# B&R Automation Studio project OpcUaSample410_BrbLibUa103 (part 8)

#### BrbIsWithinRangeUdint.c - Gibt zurück, ob sich ein Wert innerhalb eines Bereichs befindet
```c
#include <bur/plctypes.h>
#ifdef __cplusplus
	extern "C"
	{
#endif

	#include "BrbLib.h"
	#include <AnsiCFunc.h>

#ifdef __cplusplus
	};
#endif

// NOLINTBEGIN(readability-*, bugprone-easily-swappable-parameters, clang-diagnostic-invalid-utf8, clang-diagnostic-invalid-source-encoding, clang-diagnostic-pointer-arith, clang-diagnostic-strict-prototypes, hicpp-uppercase-literal-suffix, cppcoreguidelines-*, performance-*)

/* Gibt zurück, ob sich ein Wert innerhalb eines Bereichs befindet */
plcbit BrbIsWithinRangeUdint(unsigned long nValue, unsigned long nRangeMin, unsigned long nRangeMax, unsigned long nTolerance)
{
	BOOL bResult = 0;
	if(nRangeMin > nRangeMax)
	{
		UDINT nTemp = nRangeMin;
		nRangeMin = nRangeMax;
		nRangeMax = nTemp;
	}
	UDINT nMin = 0;
	if(nTolerance < nRangeMin)
	{
		nMin = nRangeMin - nTolerance;
	}
	UDINT nMax = nRangeMax + nTolerance;
	if(nValue >= nMin && nValue <= nMax)
	{
		bResult = 1;
	}
	return bResult;
}

// NOLINTEND(readability-*, bugprone-easily-swappable-parameters, clang-diagnostic-invalid-utf8, clang-diagnostic-invalid-source-encoding, clang-diagnostic-pointer-arith, clang-diagnostic-strict-prototypes, hicpp-uppercase-literal-suffix, cppcoreguidelines-*, performance-*)
```

#### BrbIsWithinRangeReal.c - Gibt zurück, ob sich ein Wert innerhalb eines Bereichs befindet
```c
#include <bur/plctypes.h>
#ifdef __cplusplus
	extern "C"
	{
#endif

	#include "BrbLib.h"
	#include <AnsiCFunc.h>

#ifdef __cplusplus
	};
#endif

// NOLINTBEGIN(readability-*, bugprone-easily-swappable-parameters, clang-diagnostic-invalid-utf8, clang-diagnostic-invalid-source-encoding, clang-diagnostic-pointer-arith, clang-diagnostic-strict-prototypes, hicpp-uppercase-literal-suffix, cppcoreguidelines-*, performance-*)

/* Gibt zurück, ob sich ein Wert innerhalb eines Bereichs befindet */
plcbit BrbIsWithinRangeReal(float rValue, float rRangeMin, float rRangeMax, float rTolerance)
{
	BOOL bResult = 0;
	if(rRangeMin > rRangeMax)
	{
		REAL nTemp = rRangeMin;
		rRangeMin = rRangeMax;
		rRangeMax = nTemp;
	}
	if(rTolerance < 0.0f)
	{
		rTolerance = rTolerance * -1.00000000000f;
	}
	REAL rMin = rRangeMin - rTolerance;
	REAL rMax = rRangeMax + rTolerance;
	if(rValue >= rMin && rValue <= rMax)
	{
		bResult = 1;
	}
	return bResult;
}

// NOLINTEND(readability-*, bugprone-easily-swappable-parameters, clang-diagnostic-invalid-utf8, clang-diagnostic-invalid-source-encoding, clang-diagnostic-pointer-arith, clang-diagnostic-strict-prototypes, hicpp-uppercase-literal-suffix, cppcoreguidelines-*, performance-*)
```

#### BrbIsWithinRangeLReal.c - Gibt zurück, ob sich ein Wert innerhalb eines Bereichs befindet
```c
#include <bur/plctypes.h>
#ifdef __cplusplus
	extern "C"
	{
#endif

	#include "BrbLib.h"
	#include <AnsiCFunc.h>

#ifdef __cplusplus
	};
#endif

// NOLINTBEGIN(readability-*, bugprone-easily-swappable-parameters, clang-diagnostic-invalid-utf8, clang-diagnostic-invalid-source-encoding, clang-diagnostic-pointer-arith, clang-diagnostic-strict-prototypes, hicpp-uppercase-literal-suffix, cppcoreguidelines-*, performance-*)

/* Gibt zurück, ob sich ein Wert innerhalb eines Bereichs befindet */
plcbit BrbIsWithinRangeLReal(double rValue, double rRangeMin, double rRangeMax, double rTolerance)
{
	BOOL bResult = 0;
	if(rRangeMin > rRangeMax)
	{
		LREAL nTemp = rRangeMin;
		rRangeMin = rRangeMax;
		rRangeMax = nTemp;
	}
	if(rTolerance < 0.0)
	{
		rTolerance = rTolerance*(LREAL)-1.00000000000;
	}
	LREAL rMin = rRangeMin - rTolerance;
	LREAL rMax = rRangeMax + rTolerance;
	if(rValue >= rMin && rValue <= rMax)
	{
		bResult = 1;
	}
	return bResult;
}

// NOLINTEND(readability-*, bugprone-easily-swappable-parameters, clang-diagnostic-invalid-utf8, clang-diagnostic-invalid-source-encoding, clang-diagnostic-pointer-arith, clang-diagnostic-strict-prototypes, hicpp-uppercase-literal-suffix, cppcoreguidelines-*, performance-*)
```

#### BrbGetAngleRad.c - Rechnet einen Winkel von Grad ins Bogenmass um
```c
/********************************************************************
 * COPYRIGHT -- Bernecker + Rainer
 ********************************************************************
 * Library: BrbLib
 * File: BrbGetAngleRad.c
 * Author: niedermeierr
 * Created: July 19, 2014
 ********************************************************************
 * Implementation of library BrbLib
 ********************************************************************/

#include <bur/plctypes.h>
#ifdef __cplusplus
	extern "C"
	{
#endif

#include "BrbLib.h"
#include <math.h>

#ifdef __cplusplus
	};
#endif

// NOLINTBEGIN(readability-*, bugprone-easily-swappable-parameters, clang-diagnostic-invalid-utf8, clang-diagnostic-invalid-source-encoding, clang-diagnostic-pointer-arith, clang-diagnostic-strict-prototypes, hicpp-uppercase-literal-suffix, cppcoreguidelines-*, performance-*)

/* Rechnet einen Winkel von Grad ins Bogenmass um */
float BrbGetAngleRad(float rAngleDeg)
{
	REAL nResult = rAngleDeg * rBRB_FACTOR_DEG_TO_RAD;
	return nResult;
}

// NOLINTEND(readability-*, bugprone-easily-swappable-parameters, clang-diagnostic-invalid-utf8, clang-diagnostic-invalid-source-encoding, clang-diagnostic-pointer-arith, clang-diagnostic-strict-prototypes, hicpp-uppercase-literal-suffix, cppcoreguidelines-*, performance-*)
```

#### BrbGetAngleDeg.c - Rechnet einen Winkel vom Bogenmass in Grad um
```c
/********************************************************************
 * COPYRIGHT -- Bernecker + Rainer
 ********************************************************************
 * Library: BrbLib
 * File: BrbGetAngleDeg.c
 * Author: niedermeierr
 * Created: July 19, 2014
 ********************************************************************
 * Implementation of library BrbLib
 ********************************************************************/

#include <bur/plctypes.h>
#ifdef __cplusplus
	extern "C"
	{
#endif

#include "BrbLib.h"
#include <math.h>

#ifdef __cplusplus
	};
#endif

// NOLINTBEGIN(readability-*, bugprone-easily-swappable-parameters, clang-diagnostic-invalid-utf8, clang-diagnostic-invalid-source-encoding, clang-diagnostic-pointer-arith, clang-diagnostic-strict-prototypes, hicpp-uppercase-literal-suffix, cppcoreguidelines-*, performance-*)

/* Rechnet einen Winkel vom Bogenmass in Grad um */
float BrbGetAngleDeg(float rAngleRad)
{
	REAL nResult = rAngleRad * rBRB_FACTOR_RAD_TO_DEG;
	return nResult;
}

// NOLINTEND(readability-*, bugprone-easily-swappable-parameters, clang-diagnostic-invalid-utf8, clang-diagnostic-invalid-source-encoding, clang-diagnostic-pointer-arith, clang-diagnostic-strict-prototypes, hicpp-uppercase-literal-suffix, cppcoreguidelines-*, performance-*)
```

#### BrbNormalizeAngleRad.c - Normalisiert einen Bogenmasswinkel in den Bereich 0..2Pi
```c
/********************************************************************
 * COPYRIGHT -- Bernecker + Rainer
 ********************************************************************
 * Library: BrbLib
 * File: BrbNormalizeAngleRad.c
 * Author: niedermeierr
 * Created: September 05, 2014
 ********************************************************************
 * Implementation of library BrbLib
 ********************************************************************/

#include <bur/plctypes.h>
#ifdef __cplusplus
	extern "C"
	{
#endif

#include "BrbLib.h"
#include <AnsiCFunc.h>

#ifdef __cplusplus
	};
#endif

// NOLINTBEGIN(readability-*, bugprone-easily-swappable-parameters, clang-diagnostic-invalid-utf8, clang-diagnostic-invalid-source-encoding, clang-diagnostic-pointer-arith, clang-diagnostic-strict-prototypes, hicpp-uppercase-literal-suffix, cppcoreguidelines-*, performance-*)

/* Normalisiert einen Bogenmass-Winkel in den Bereich 0..2Pi */
float BrbNormalizeAngleRad(float rAngleRad)
{
	REAL rResult = 0.0f;
	DINT nMod = (DINT)(rAngleRad / 6.283185307179586476925286766559f);
	rResult = rAngleRad - ((REAL)nMod * 6.283185307179586476925286766559f);
	if(BrbIsNearlyZeroReal(rResult, 0.00017453292519943f))
	{
		// ~= 0.0
		rResult = 0.0f;
	}
	else if(rResult < 0.0f)
	{
		rResult += 6.283185307179586476925286766559f;
	}
	return rResult;
}

// NOLINTEND(readability-*, bugprone-easily-swappable-parameters, clang-diagnostic-invalid-utf8, clang-diagnostic-invalid-source-encoding, clang-diagnostic-pointer-arith, clang-diagnostic-strict-prototypes, hicpp-uppercase-literal-suffix, cppcoreguidelines-*, performance-*)
```

#### BrbNormalizeAngleDeg.c - Normalisiert einen Grad-Winkel in den Bereich 0..360°
```c
/********************************************************************
 * COPYRIGHT -- Bernecker + Rainer
 ********************************************************************
 * Library: BrbLib
 * File: BrbNormalizeAngleDeg.c
 * Author: niedermeierr
 * Created: September 05, 2014
 ********************************************************************
 * Implementation of library BrbLib
 ********************************************************************/

#include <bur/plctypes.h>
#ifdef __cplusplus
	extern "C"
	{
#endif

	#include "BrbLib.h"

#ifdef __cplusplus
	};
#endif

// NOLINTBEGIN(readability-*, bugprone-easily-swappable-parameters, clang-diagnostic-invalid-utf8, clang-diagnostic-invalid-source-encoding, clang-diagnostic-pointer-arith, clang-diagnostic-strict-prototypes, hicpp-uppercase-literal-suffix, cppcoreguidelines-*, performance-*)

/* Normalisiert einen Grad-Winkel in den Bereich 0..360° */
float BrbNormalizeAngleDeg(float rAngleDeg, plcbit bKeep360)
{
	REAL rResult = rBRB_DEGREE_0;
	if(bKeep360 == 1 && rAngleDeg == rBRB_DEGREE_360)
	{
		// 360.0° ist eigentlich 0°. Diese Korrektur kann hier verhindert werden.
		rResult = rBRB_DEGREE_360;
	}
	else
	{
		DINT nMod = (DINT)(rAngleDeg / rBRB_DEGREE_360);
		rResult = rAngleDeg - ((REAL)nMod * rBRB_DEGREE_360);
		if(rResult < rBRB_DEGREE_0)
		{
			rResult += rBRB_DEGREE_360;
		}
	}
	return rResult;
}

// NOLINTEND(readability-*, bugprone-easily-swappable-parameters, clang-diagnostic-invalid-utf8, clang-diagnostic-invalid-source-encoding, clang-diagnostic-pointer-arith, clang-diagnostic-strict-prototypes, hicpp-uppercase-literal-suffix, cppcoreguidelines-*, performance-*)
```

#### BrbIsWithinRangeAngle.c - Gibt zurück, ob sich ein Winkel innerhalb eines Bereichs befindet
```c
#include <bur/plctypes.h>
#ifdef __cplusplus
	extern "C"
	{
#endif

#include "BrbLib.h"

#ifdef __cplusplus
	};
#endif

// NOLINTBEGIN(readability-*, bugprone-easily-swappable-parameters, clang-diagnostic-invalid-utf8, clang-diagnostic-invalid-source-encoding, clang-diagnostic-pointer-arith, clang-diagnostic-strict-prototypes, hicpp-uppercase-literal-suffix, cppcoreguidelines-*, performance-*)

/* Gibt zurück, ob sich ein Winkel innerhalb eines Bereichs befindet */
plcbit BrbIsWithinRangeAngle(double rAngleAct, double rAngleStart, double rAngleEnd)
{
	BOOL bResult = 0;
	if(rAngleStart <= rAngleEnd)
	{
		if(rAngleAct >= rAngleStart && rAngleAct <= rAngleEnd)
		{
			bResult = 1;
		}
	}
	else
	{
		if(rAngleAct >= rAngleStart || rAngleAct <= rAngleEnd)
		{
			bResult = 1;
		}
	}
	return bResult;
}

// NOLINTEND(readability-*, bugprone-easily-swappable-parameters, clang-diagnostic-invalid-utf8, clang-diagnostic-invalid-source-encoding, clang-diagnostic-pointer-arith, clang-diagnostic-strict-prototypes, hicpp-uppercase-literal-suffix, cppcoreguidelines-*, performance-*)
```

#### BrbDetectAngleTransition.c - Erkennt eine Winkel-Übergang
```c
#include <bur/plctypes.h>
#ifdef __cplusplus
	extern "C"
	{
#endif

#include "BrbLib.h"

#ifdef __cplusplus
	};
#endif

// NOLINTBEGIN(readability-*, bugprone-easily-swappable-parameters, clang-diagnostic-invalid-utf8, clang-diagnostic-invalid-source-encoding, clang-diagnostic-pointer-arith, clang-diagnostic-strict-prototypes, hicpp-uppercase-literal-suffix, cppcoreguidelines-*, performance-*)

/* Erkennt den Übergang einer bestimmten Position bei einer 360°-Rundachse */
plcbit BrbDetectAngleTransition(double rTransPosition, plcbit bDirection, double rPosAct, double rPosOld)
{
	BOOL bResult = 0;
	// Richtung feststellen
	LREAL rDir =  rPosAct - rPosOld;
	if(rPosAct >= rBRB_DEGREE_0 && rPosAct <= rBRB_DEGREE_90 && rPosOld >= rBRB_DEGREE_270 && rPosOld <= rBRB_DEGREE_360)
	{
		// Übergang von 360° auf 0°
		rDir = +1.0;
	}
	else if(rPosAct >= rBRB_DEGREE_270 && rPosAct <= rBRB_DEGREE_360 && rPosOld >= rBRB_DEGREE_0 && rPosOld <= rBRB_DEGREE_90)
	{
		// Übergang von 0° auf 360°
		rDir = -1.0;
	}
	if(rTransPosition <= rBRB_DEGREE_90)
	{
		// Positionen um 90° nach positiv verschieben, um Übergang von 360° auf 0° zu vermeiden
		rTransPosition = (LREAL)BrbNormalizeAngleDeg((REAL)rTransPosition + rBRB_DEGREE_90, 0);
		rPosAct = (LREAL)BrbNormalizeAngleDeg((REAL)rPosAct + rBRB_DEGREE_90, 0);
		rPosOld = (LREAL)BrbNormalizeAngleDeg((REAL)rPosOld + rBRB_DEGREE_90, 0);
	}
	else if(rTransPosition >= rBRB_DEGREE_270)
	{
		// Positionen um 90° nach negativ verschieben, um Übergang von 360° auf 0° zu vermeiden
		rTransPosition = (LREAL)BrbNormalizeAngleDeg((REAL)rTransPosition - rBRB_DEGREE_90, 0);
		rPosAct = (LREAL)BrbNormalizeAngleDeg((REAL)rPosAct - rBRB_DEGREE_90, 0);
		rPosOld = (LREAL)BrbNormalizeAngleDeg((REAL)rPosOld - rBRB_DEGREE_90, 0);
	}
	// NOLINTBEGIN(bugprone-branch-clone)
	if(bDirection == 0 && rDir < rBRB_DEGREE_0)
	{
		// Negative Richtung
		if(rPosOld > rTransPosition && rPosAct <= rTransPosition)
		{
			bResult = 1;
		}
		else if(rPosOld >= rTransPosition && rPosAct < rTransPosition)
		{
			bResult = 1;
		}
	}
	else if(bDirection == 1 && rDir > rBRB_DEGREE_0)
	{
		// Positive Richtung
		if(rPosOld < rTransPosition && rPosAct >= rTransPosition)
		{
			bResult = 1;
		}
		else if(rPosOld <= rTransPosition && rPosAct > rTransPosition)
		{
			bResult = 1;
		}
	}
	// NOLINTEND(bugprone-branch-clone)
	return bResult;
}

// NOLINTEND(readability-*, bugprone-easily-swappable-parameters, clang-diagnostic-invalid-utf8, clang-diagnostic-invalid-source-encoding, clang-diagnostic-pointer-arith, clang-diagnostic-strict-prototypes, hicpp-uppercase-literal-suffix, cppcoreguidelines-*, performance-*)
```

#### BrbGetDistance2d.c - Errechnet die Distanz zwischen zwei Punkten
```c
#include <bur/plctypes.h>
#ifdef __cplusplus
	extern "C"
	{
#endif

	#include "BrbLib.h"
	#include <math.h>

#ifdef __cplusplus
	};
#endif

// NOLINTBEGIN(readability-*, bugprone-easily-swappable-parameters, clang-diagnostic-invalid-utf8, clang-diagnostic-invalid-source-encoding, clang-diagnostic-pointer-arith, clang-diagnostic-strict-prototypes, hicpp-uppercase-literal-suffix, cppcoreguidelines-*, performance-*)

/* Gibt die Distanz zwischen zwei Punkten im 2-dimensionalen Raum zurück */
double BrbGetDistance2d(double rX1, double rY1, double rX2, double rY2)
{
	return sqrt(pow((rX1-rX2), 2) + pow((rY1-rY2), 2));
}

// NOLINTEND(readability-*, bugprone-easily-swappable-parameters, clang-diagnostic-invalid-utf8, clang-diagnostic-invalid-source-encoding, clang-diagnostic-pointer-arith, clang-diagnostic-strict-prototypes, hicpp-uppercase-literal-suffix, cppcoreguidelines-*, performance-*)
```

#### BrbRoundDint.c - Rundet einen Dint
```c
/********************************************************************
 * COPYRIGHT -- Bernecker + Rainer
 ********************************************************************
 * Library: BrbLib
 * File: BrbRoundDint.c
 * Author: niedermeierr
 * Created: November 19, 2015
 ********************************************************************
 * Implementation of library BrbLib
 ********************************************************************/

#include <bur/plctypes.h>
#ifdef __cplusplus
	extern "C"
	{
#endif

#include "BrbLib.h"
#include <math.h>

#ifdef __cplusplus
	};
#endif

// NOLINTBEGIN(readability-*, bugprone-easily-swappable-parameters, clang-diagnostic-invalid-utf8, clang-diagnostic-invalid-source-encoding, clang-diagnostic-pointer-arith, clang-diagnostic-strict-prototypes, hicpp-uppercase-literal-suffix, cppcoreguidelines-*, performance-*)

/* Rundet einen Dint */
signed long BrbRoundDint(signed long nValue, enum BrbRound_ENUM eRound, unsigned char nDigits) // NOLINT(readability-function-cognitive-complexity)
{
	DINT nResult = nValue;
	if(nValue != 0)
	{
		if(nDigits < 1)
		{
			nDigits = 1;
		}
		BOOL bMinus = 0;
		if(nValue < 0)
		{
			bMinus = 1;
			nResult = nResult * -1;
			if(eRound == eBRB_ROUND_UP)
			{
				eRound = eBRB_ROUND_DOWN;
			}
			else if(eRound == eBRB_ROUND_DOWN)
			{
				eRound = eBRB_ROUND_UP;
			}
		}
		if(eRound == eBRB_ROUND_UP)
		{
			// Jede Stelle für sich runden
			USINT nDigit = 0;
			for(nDigit=1; nDigit<=nDigits; nDigit++)
			{
				DINT nDigitFactor = (DINT)pow(10, nDigit); // NOLINT(clang-diagnostic-bad-function-cast)
				DINT nNum0 = (DINT)((nResult / nDigitFactor) * nDigitFactor);
				DINT nRest = nResult - nNum0;
				if(nRest > 0)
				{
					nResult = nResult + (nDigitFactor - nRest);
				}
			}
		}
		else if(eRound == eBRB_ROUND_DOWN)
		{
			// Alle Rundungs-Stellen auf 0 setzen
			DINT nDigitFactor = (DINT)pow(10, nDigits); // NOLINT(clang-diagnostic-bad-function-cast)
			DINT nNum0 = (DINT)((nResult / nDigitFactor) * nDigitFactor);
			DINT nRest = nResult - nNum0;
			nResult = nResult - nRest;
		}
		else
		{
			DINT nDigitFactor = (DINT)pow(10.0, nDigits); // NOLINT(clang-diagnostic-bad-function-cast)
			DINT nNum0 = (DINT)(nResult / nDigitFactor);
			DINT nNum1 = nNum0 * nDigitFactor;
			DINT nRest = nResult - nNum1; // Rundungs-Stelle feststellen
			if(nRest >= 5 * (DINT)(nDigitFactor / 10.0))
			{
				nResult = BrbRoundDint(nResult, eBRB_ROUND_UP, nDigits);
			}
			else
			{
				nResult = BrbRoundDint(nResult, eBRB_ROUND_DOWN, nDigits);
			}
		}
		if(bMinus == 1)
		{
			nResult = nResult * -1;
		}
	}
	return nResult;
}

// NOLINTEND(readability-*, bugprone-easily-swappable-parameters, clang-diagnostic-invalid-utf8, clang-diagnostic-invalid-source-encoding, clang-diagnostic-pointer-arith, clang-diagnostic-strict-prototypes, hicpp-uppercase-literal-suffix, cppcoreguidelines-*, performance-*)
```

#### BrbScaleLReal.c - Skaliert ein analoges Eingangssignal linear auf einen Einheitswert
```c
/********************************************************************
 * COPYRIGHT -- Bernecker + Rainer
 ********************************************************************
 * Library: BrbLib
 * File: BrbScaleLReal.c
 * Author: niedermeierr
 * Created: October 11, 2021
 ********************************************************************
 * Implementation of library BrbLib
 ********************************************************************/

#include <bur/plctypes.h>
#ifdef __cplusplus
	extern "C"
	{
#endif

#include "BrbLib.h"

#ifdef __cplusplus
	};
#endif

// NOLINTBEGIN(readability-*, bugprone-easily-swappable-parameters, clang-diagnostic-invalid-utf8, clang-diagnostic-invalid-source-encoding, clang-diagnostic-pointer-arith, clang-diagnostic-strict-prototypes, hicpp-uppercase-literal-suffix, cppcoreguidelines-*, performance-*)

/* Skaliert ein analoges Signal linear */
double BrbScaleLReal(double rRaw, double rRawMin, double rRawMax, double rScaledMin, double rScaledMax, double rFactor, double rOffset)
{
	LREAL rResult = 0.0;
	LREAL rRawDiff = rRawMax - rRawMin;
	if(rRawDiff != 0.0) // Division durch 0 vermeiden
	{
		rResult = ((rScaledMin + ((rScaledMax - rScaledMin) / rRawDiff * (rRaw - rRawMin))) * rFactor) + rOffset;
	}
	return rResult;
}

// NOLINTEND(readability-*, bugprone-easily-swappable-parameters, clang-diagnostic-invalid-utf8, clang-diagnostic-invalid-source-encoding, clang-diagnostic-pointer-arith, clang-diagnostic-strict-prototypes, hicpp-uppercase-literal-suffix, cppcoreguidelines-*, performance-*)
```

#### BrbScaleAnalogInput.c - Skaliert ein analoges Eingangssignal linear auf einen Einheitswert
```c
/********************************************************************
 * COPYRIGHT -- Bernecker + Rainer
 ********************************************************************
 * Library: BrbLib
 * File: BrbScaleAnalogInput.c
 * Author: niedermeierr
 * Created: April 22, 2016
 ********************************************************************
 * Implementation of library BrbLib
 ********************************************************************/

#include <bur/plctypes.h>
#ifdef __cplusplus
	extern "C"
	{
#endif

#include "BrbLib.h"

#ifdef __cplusplus
	};
#endif

// NOLINTBEGIN(readability-*, bugprone-easily-swappable-parameters, clang-diagnostic-invalid-utf8, clang-diagnostic-invalid-source-encoding, clang-diagnostic-pointer-arith, clang-diagnostic-strict-prototypes, hicpp-uppercase-literal-suffix, cppcoreguidelines-*, performance-*)

/* Skaliert ein analoges Eingangssignal linear auf einen Einheitswert */
float BrbScaleAnalogInput(signed short nRaw, signed short nRawMin, signed short nRawMax, float rScaledMin, float rScaledMax, float rFactor, float rOffset)
{
	REAL rResult = 0.0f;
	DINT nRawDiff = nRawMax - nRawMin;
	if(nRawDiff != 0) // Division durch 0 vermeiden
	{
		rResult = ((rScaledMin + ((rScaledMax - rScaledMin) / (REAL)nRawDiff * (REAL)(nRaw - nRawMin))) * rFactor) + rOffset;
	}
	return rResult;
}

// NOLINTEND(readability-*, bugprone-easily-swappable-parameters, clang-diagnostic-invalid-utf8, clang-diagnostic-invalid-source-encoding, clang-diagnostic-pointer-arith, clang-diagnostic-strict-prototypes, hicpp-uppercase-literal-suffix, cppcoreguidelines-*, performance-*)
```

#### BrbScaleAnalogOutput.c - Skaliert ein analoges Ausgangssignal von einem EInheitswert
```c
/********************************************************************
 * COPYRIGHT -- Bernecker + Rainer
 ********************************************************************
 * Library: BrbLib
 * File: BrbScaleAnalogOutput.c
 * Author: niedermeierr
 * Created: April 22, 2016
 ********************************************************************
 * Implementation of library BrbLib
 ********************************************************************/

#include <bur/plctypes.h>
#ifdef __cplusplus
	extern "C"
	{
#endif

#include "BrbLib.h"

#ifdef __cplusplus
	};
#endif

// NOLINTBEGIN(readability-*, bugprone-easily-swappable-parameters, clang-diagnostic-invalid-utf8, clang-diagnostic-invalid-source-encoding, clang-diagnostic-pointer-arith, clang-diagnostic-strict-prototypes, hicpp-uppercase-literal-suffix, cppcoreguidelines-*, performance-*)

/* Skaliert ein analoges Ausgangssignal von einem Einheitswert */
signed short BrbScaleAnalogOutput(float rScaled, signed short nRawMin, signed short nRawMax, float rScaledMin, float rScaledMax, float rFactor, float rOffset)
{
	INT nResult = 0;
	REAL rScaleDiff = (rScaledMax - rScaledMin);
	if(rFactor != 0.0f && rScaleDiff != 0.0f) // Division durch 0 vermeiden // NOLINT(clang-diagnostic-float-equal)
	{
		REAL rRawMin = (REAL)nRawMin;
		REAL rRawMax = (REAL)nRawMax;
		REAL rValue = ((((rScaled - rOffset) / rFactor) - rScaledMin) * (rRawMax - rRawMin) / rScaleDiff) + rRawMin;
		if(rValue < rRawMin)
		{
			nResult = nRawMin;
		}
		else if(rValue > rRawMax)
		{
			nResult = nRawMax;
		}
		else
		{
			nResult = (INT)rValue;
		}
	}
	return nResult;
}

// NOLINTEND(readability-*, bugprone-easily-swappable-parameters, clang-diagnostic-invalid-utf8, clang-diagnostic-invalid-source-encoding, clang-diagnostic-pointer-arith, clang-diagnostic-strict-prototypes, hicpp-uppercase-literal-suffix, cppcoreguidelines-*, performance-*)
```

#### Package Logical/Libraries/BrbLib/Random - Erzeugung von Zufalls-Werten

#### BrbGetRandomPercent.c - Erzeugt eine Zufallszahl zwischen 0.0 und 1.0
```c
/********************************************************************
 * COPYRIGHT -- Bernecker + Rainer
 ********************************************************************
 * Library: BrbLib
 * File: BrbGetRandomPercent.c
 * Author: niedermeierr
 * Created: June 11, 2013
 ********************************************************************
 * Implementation of library BrbLib
 ********************************************************************/

#include <bur/plctypes.h>
#ifdef __cplusplus
	extern "C"
	{
#endif

#include "BrbLib.h"
#include "AnsiCFunc.h"

#ifdef __cplusplus
	};
#endif

// NOLINTBEGIN(readability-*, bugprone-easily-swappable-parameters, clang-diagnostic-invalid-utf8, clang-diagnostic-invalid-source-encoding, clang-diagnostic-pointer-arith, clang-diagnostic-strict-prototypes, hicpp-uppercase-literal-suffix, cppcoreguidelines-*, performance-*)

/* Erzeugt eine Zufallszahl zwischen 0.0 und 1.0 */
float BrbGetRandomPercent()
{
	INT	 	nRandom1 = (INT)rand(); // NOLINT(cert-msc30-c,cert-msc50-cpp, concurrency-mt-unsafe)
	DINT	nRandom2 = (DINT)nRandom1 + 32768;
	REAL	rRandom3 = (REAL)nRandom2 / 65535.0f;
	return rRandom3;
}

// NOLINTEND(readability-*, bugprone-easily-swappable-parameters, clang-diagnostic-invalid-utf8, clang-diagnostic-invalid-source-encoding, clang-diagnostic-pointer-arith, clang-diagnostic-strict-prototypes, hicpp-uppercase-literal-suffix, cppcoreguidelines-*, performance-*)
```

#### BrbGetRandomBool.c - Erzeugt einen boolschen Zufallswert
```c
/********************************************************************
 * COPYRIGHT -- Bernecker + Rainer
 ********************************************************************
 * Library: BrbLib
 * File: BrbGetRandomBool.c
 * Author: niedermeierr
 * Created: June 11, 2013
 ********************************************************************
 * Implementation of library BrbLib
 ********************************************************************/

#include <bur/plctypes.h>
#ifdef __cplusplus
	extern "C"
	{
#endif

#include "BrbLib.h"

#ifdef __cplusplus
	};
#endif

// NOLINTBEGIN(readability-*, bugprone-easily-swappable-parameters, clang-diagnostic-invalid-utf8, clang-diagnostic-invalid-source-encoding, clang-diagnostic-pointer-arith, clang-diagnostic-strict-prototypes, hicpp-uppercase-literal-suffix, cppcoreguidelines-*, performance-*)

/* Erzeugt einen boolschen Zufallswert */
plcbit BrbGetRandomBool()
{
	BOOL bRandom = (BOOL)(BrbGetRandomPercent()*(2));
	return bRandom;
}

// NOLINTEND(readability-*, bugprone-easily-swappable-parameters, clang-diagnostic-invalid-utf8, clang-diagnostic-invalid-source-encoding, clang-diagnostic-pointer-arith, clang-diagnostic-strict-prototypes, hicpp-uppercase-literal-suffix, cppcoreguidelines-*, performance-*)
```

#### BrbGetRandomUdint.c - Erzeugt eine Zufallszahl zwischen nMin und nMax
```c
/********************************************************************
 * COPYRIGHT -- Bernecker + Rainer
 ********************************************************************
 * Library: BrbLib
 * File: BrbGetRandomUdint.c
 * Author: niedermeierr
 * Created: June 11, 2013
 ********************************************************************
 * Implementation of library BrbLib
 ********************************************************************/

#include <bur/plctypes.h>
#ifdef __cplusplus
	extern "C"
	{
#endif

#include "BrbLib.h"

#ifdef __cplusplus
	};
#endif

// NOLINTBEGIN(readability-*, bugprone-easily-swappable-parameters, clang-diagnostic-invalid-utf8, clang-diagnostic-invalid-source-encoding, clang-diagnostic-pointer-arith, clang-diagnostic-strict-prototypes, hicpp-uppercase-literal-suffix, cppcoreguidelines-*, performance-*)

/* Erzeugt eine Zufallszahl zwischen nMin und nMax */
unsigned long BrbGetRandomUdint(unsigned long nMin, unsigned long nMax)
{
	UDINT nRandom = 0;
	if(nMin == 0 && nMax == nBRB_UDINT_MAX)
	{
		nRandom = (UDINT)(BrbGetRandomPercent() * (REAL)nMax);
	}
	else
	{
		// Eigentlich ohne +1, aber dann ist es sehr unwahrscheinlich, dass sich der Max-Wert ergibt (RandomPercent muss 1.0 sein).
		// Das +1 erhöht die Chance dazu, muss dann aber korrigiert werden.
		nRandom = (UDINT)(BrbGetRandomPercent()*(REAL)(nMax-nMin+1))+nMin;
		if(nRandom > nMax)
		{
			nRandom = nMax;
		}
		else if(nMin > 0 && nMax == nBRB_UDINT_MAX && nRandom == 0)
		{
			nRandom = nBRB_UDINT_MAX;
		}
	}
	return nRandom;
}

// NOLINTEND(readability-*, bugprone-easily-swappable-parameters, clang-diagnostic-invalid-utf8, clang-diagnostic-invalid-source-encoding, clang-diagnostic-pointer-arith, clang-diagnostic-strict-prototypes, hicpp-uppercase-literal-suffix, cppcoreguidelines-*, performance-*)
```

#### BrbGetRandomDint.c - Erzeugt eine Zufallszahl zwischen nMin und nMax
```c
/********************************************************************
 * COPYRIGHT -- Bernecker + Rainer
 ********************************************************************
 * Library: BrbLib
 * File: BrbGetRandomDint.c
 * Author: niedermeierr
 * Created: June 11, 2013
 ********************************************************************
 * Implementation of library BrbLib
 ********************************************************************/

#include <bur/plctypes.h>
#ifdef __cplusplus
	extern "C"
	{
#endif

#include "BrbLib.h"
#include <AnsiCFunc.h>

#ifdef __cplusplus
	};
#endif

// NOLINTBEGIN(readability-*, bugprone-easily-swappable-parameters, clang-diagnostic-invalid-utf8, clang-diagnostic-invalid-source-encoding, clang-diagnostic-pointer-arith, clang-diagnostic-strict-prototypes, hicpp-uppercase-literal-suffix, cppcoreguidelines-*, performance-*)

/* Erzeugt eine Zufallszahl zwischen nMin und nMax */
signed long BrbGetRandomDint(signed long nMin, signed long nMax)
{
	DINT nRandom = 0;
	if(nMin >= 0 && nMax >= 0)
	{
		nRandom = (DINT)BrbGetRandomUdint((UDINT)nMin, (UDINT)nMax);
	}
	else if(nMin < 0 && nMax < 0)
	{
		nRandom = (DINT)BrbGetRandomUdint((UDINT)abs(nMax), (UDINT)abs(nMin));
		nRandom = nRandom * -1;
	}
	else
	{
		// Eigentlich ohne +2.0, aber dann ist es sehr unwahrscheinlich, dass sich der Max-Wert ergibt (RandomPercent muss 1.0 sein).
		// Das +2.0 erhöht die Chance dazu, muss dann aber korrigiert werden.
		LREAL rRange = (LREAL)nMax - (LREAL)nMin + (LREAL)2.0;
		REAL rRangeRandom = BrbGetRandomPercent() * (REAL)rRange;
		LREAL rRandom = (LREAL)rRangeRandom + (LREAL)nMin - (LREAL)1.0;
		nRandom = (DINT)rRandom;
		// NOLINTBEGIN(bugprone-branch-clone)
		if(nRandom > nMax)
		{
			nRandom = nMax;
		}
		else if(nMin > 0 && nMax == nBRB_DINT_MAX && nRandom == 0)
		{
			nRandom = nMax;
		}
		else if(nRandom < nMin)
		{
			nRandom = nMin;
		}
		// NOLINTEND(bugprone-branch-clone)
	}
	return nRandom;
}

// NOLINTEND(readability-*, bugprone-easily-swappable-parameters, clang-diagnostic-invalid-utf8, clang-diagnostic-invalid-source-encoding, clang-diagnostic-pointer-arith, clang-diagnostic-strict-prototypes, hicpp-uppercase-literal-suffix, cppcoreguidelines-*, performance-*)
```

#### BrbGetRandomText.c - Erzeugt einen Zufallstext mit bestimmter Länge (nur Zahlen, Groß- und Kleinbuchstaben)
```c
#include <bur/plctypes.h>
#ifdef __cplusplus
	extern "C"
	{
#endif
	#include "BrbLib.h"
#include <string.h>

#ifdef __cplusplus
	};
#endif

// NOLINTBEGIN(readability-*, bugprone-easily-swappable-parameters, clang-diagnostic-invalid-utf8, clang-diagnostic-invalid-source-encoding, clang-diagnostic-pointer-arith, clang-diagnostic-strict-prototypes, hicpp-uppercase-literal-suffix, cppcoreguidelines-*, performance-*)

/* Erzeugt einen Zufallstext mit bestimmter Länge (nur Zahlen, Groß- und Kleinbuchstaben) */
unsigned long BrbGetRandomText(plcstring* pText, unsigned long nTextSize, unsigned long nTextLength)
{
	memset(pText, 0, nTextSize);
	if(nTextLength >= nTextSize)
	{
		nTextLength = nTextSize-1;
	}
	UDINT nCharIndex = 0;
	for(nCharIndex=0; nCharIndex<nTextLength; nCharIndex++)
	{
		USINT nChar = 0;
		DINT nBlockIndex = BrbGetRandomDint(0,2);
		if (nBlockIndex == 0)
		{
			// Zahl
			nChar = (USINT)BrbGetRandomUdint(48,57);
		}
		else if (nBlockIndex == 1)
		{
			// Großbuchstabe
			nChar = (USINT)BrbGetRandomUdint(65,90);
		}
		else
		{
			// KLeinbuchstabe
			nChar = (USINT)BrbGetRandomUdint(97,122);
		}
		USINT* pChar = (USINT*)pText + nCharIndex;
		*pChar = nChar;
	}
	return nTextLength;
}

// NOLINTEND(readability-*, bugprone-easily-swappable-parameters, clang-diagnostic-invalid-utf8, clang-diagnostic-invalid-source-encoding, clang-diagnostic-pointer-arith, clang-diagnostic-strict-prototypes, hicpp-uppercase-literal-suffix, cppcoreguidelines-*, performance-*)
```

#### BrbGetRandomString.c - Erzeugt einen Zufallstext mit bestimmter Länge aus einer Blockauswahl
```c
#include <bur/plctypes.h>
#ifdef __cplusplus
	extern "C"
	{
#endif
	#include "BrbLib.h"
	#include <string.h>

#ifdef __cplusplus
	};
#endif

// NOLINTBEGIN(readability-*, bugprone-easily-swappable-parameters, clang-diagnostic-invalid-utf8, clang-diagnostic-invalid-source-encoding, clang-diagnostic-pointer-arith, clang-diagnostic-strict-prototypes, hicpp-uppercase-literal-suffix, cppcoreguidelines-*, performance-*)

/* Erzeugt einen Zufallstext mit bestimmter Länge aus einer Zeichenblockauswahl */
unsigned long BrbGetRandomString(plcstring* pText, unsigned long nTextSize, unsigned long nTextLength, enum BrbRandomString_ENUM eSelection)
{
	USINT anSelection[256];
	memset((USINT*)&anSelection, 0, sizeof(anSelection));
	UINT nChar = 0;
	UINT nSelectionLength = 0;
	if((eSelection & eBRB_RANDOM_STRING_NUMBERS) == eBRB_RANDOM_STRING_NUMBERS) // NOLINT(hicpp-signed-bitwise)
	{
		// 0123456789
		for(nChar=48;nChar<=57;nChar++)
		{
			anSelection[nSelectionLength] = (USINT)nChar;
			nSelectionLength++;
		}
	}
	if((eSelection & eBRB_RANDOM_STRING_UPPER_LETTERS) == eBRB_RANDOM_STRING_UPPER_LETTERS) // NOLINT(hicpp-signed-bitwise)
	{
		//ABCDEFGHIJKLMNOPQRSTUVWXYZ
		for(nChar=65;nChar<=90;nChar++)
		{
			anSelection[nSelectionLength] = (USINT)nChar;
			nSelectionLength++;
		}
	}
	if((eSelection & eBRB_RANDOM_STRING_LOWER_LETTERS) == eBRB_RANDOM_STRING_LOWER_LETTERS) // NOLINT(hicpp-signed-bitwise)
	{
		//abcdefghijklmnopqrstuvwxyz
		for(nChar=97;nChar<=122;nChar++)
		{
			anSelection[nSelectionLength] = (USINT)nChar;
			nSelectionLength++;
		}
	}
	if((eSelection & eBRB_RANDOM_STRING_SPACE) == eBRB_RANDOM_STRING_SPACE) // NOLINT(hicpp-signed-bitwise)
	{
		//" "
		anSelection[nSelectionLength] = 32;
		nSelectionLength++;
	}
	if((eSelection & eBRB_RANDOM_STRING_PUNCTUATION) == eBRB_RANDOM_STRING_PUNCTUATION) // NOLINT(hicpp-signed-bitwise)
	{
		//!"#$%&'()*+,-./
		for(nChar=33;nChar<=47;nChar++)
		{
			anSelection[nSelectionLength] = (USINT)nChar;
			nSelectionLength++;
		}
		//:;<=>?@
		for(nChar=58;nChar<=64;nChar++)
		{
			anSelection[nSelectionLength] = (USINT)nChar;
			nSelectionLength++;
		}
		//[\]^_`
		for(nChar=91;nChar<=96;nChar++)
		{
			anSelection[nSelectionLength] = (USINT)nChar;
			nSelectionLength++;
		}
		// {|}~
		for(nChar=123;nChar<=126;nChar++)
		{
			anSelection[nSelectionLength] = (USINT)nChar;
			nSelectionLength++;
		}
	}
	if((eSelection & eBRB_RANDOM_STRING_SYMBOLS) == eBRB_RANDOM_STRING_SYMBOLS) // NOLINT(hicpp-signed-bitwise)
	{
		for(nChar=128;nChar<=255;nChar++)
		{
			anSelection[nSelectionLength] = (USINT)nChar;
			nSelectionLength++;
		}
	}
	if((eSelection & eBRB_RANDOM_STRING_CONTROLCHARS) == eBRB_RANDOM_STRING_CONTROLCHARS) // NOLINT(hicpp-signed-bitwise)
	{
		// <127=DEL>
		anSelection[nSelectionLength] = 127;
		nSelectionLength++;
		// <1=SOH><2=STX><3=ETX><4=EOT><5=ENQ><6=ACK><7=BEL><8=BS><9=TAB><10=LF><11=VT><12=FF><13=CR><14=SO><15=SI><16=DLE>
		// <17=DC1><18=DC2><19=DC3><20=DC4><21=NAK><22=SYN><23=ETB><24=CAN><25=EM><26=SUB>27=ESC<28=FS><29=GS><30=RS><31=US>
		for(nChar=1;nChar<=31;nChar++)
		{
			anSelection[nSelectionLength] = (USINT)nChar;
			nSelectionLength++;
		}
	}
	return BrbGetRandomStringExt(pText, nTextSize, nTextLength, (STRING*)&anSelection);
}

// NOLINTEND(readability-*, bugprone-easily-swappable-parameters, clang-diagnostic-invalid-utf8, clang-diagnostic-invalid-source-encoding, clang-diagnostic-pointer-arith, clang-diagnostic-strict-prototypes, hicpp-uppercase-literal-suffix, cppcoreguidelines-*, performance-*)
```

#### BrbGetRandomStringExt.c - Erzeugt einen Zufallstext mit bestimmter Länge aus einer Zeichenauswahl
```c
#include <bur/plctypes.h>
#ifdef __cplusplus
	extern "C"
	{
#endif
	#include "BrbLib.h"
	#include <string.h>

#ifdef __cplusplus
	};
#endif

// NOLINTBEGIN(readability-*, bugprone-easily-swappable-parameters, clang-diagnostic-invalid-utf8, clang-diagnostic-invalid-source-encoding, clang-diagnostic-pointer-arith, clang-diagnostic-strict-prototypes, hicpp-uppercase-literal-suffix, cppcoreguidelines-*, performance-*)

/* Erzeugt einen Zufallstext mit bestimmter Länge aus einer Zeichenauswahl */
unsigned long BrbGetRandomStringExt(plcstring* pText, unsigned long nTextSize, unsigned long nTextLength, plcstring* pSelection)
{
	memset(pText, 0, nTextSize);
	UDINT nSelectionLength = strlen(pSelection);
	if(nSelectionLength > 0)
	{
		if(nTextLength >= nTextSize)
		{
			nTextLength = nTextSize-1;
		}
		UDINT nCharIndex = 0;
		for(nCharIndex=0; nCharIndex<nTextLength; nCharIndex++)
		{
			UDINT nSelectionCharIndex = BrbGetRandomUdint(0,nSelectionLength-1);
			USINT* pChar = (USINT*)pText + nCharIndex;
			*pChar = *((USINT*)pSelection + nSelectionCharIndex);
		}
	}
	else
	{
		nTextLength = 0;
	}
	return nTextLength;
}

// NOLINTEND(readability-*, bugprone-easily-swappable-parameters, clang-diagnostic-invalid-utf8, clang-diagnostic-invalid-source-encoding, clang-diagnostic-pointer-arith, clang-diagnostic-strict-prototypes, hicpp-uppercase-literal-suffix, cppcoreguidelines-*, performance-*)
```

#### Package Logical/Libraries/BrbLib/IpAndSubnet - Ip-Adress-Funktionen

#### BrbIpToNumericalArray.c - Wandelt eine Ip-Adresse in eine Byte-Array
```c
/********************************************************************
 * COPYRIGHT -- Bernecker + Rainer
 ********************************************************************
 * Library: BrbLib
 * File: BrbIpToNumericalArray.c
 * Author: niedermeierr
 * Created: July 05, 2022
 ********************************************************************
 * Implementation of library BrbLib
 ********************************************************************/

#include <bur/plctypes.h>
#ifdef __cplusplus
	extern "C"
	{
#endif

#include "BrbLib.h"
#include <string.h>

#ifdef __cplusplus
	};
#endif

// NOLINTBEGIN(readability-*, bugprone-easily-swappable-parameters, clang-diagnostic-invalid-utf8, clang-diagnostic-invalid-source-encoding, clang-diagnostic-pointer-arith, clang-diagnostic-strict-prototypes, hicpp-uppercase-literal-suffix, cppcoreguidelines-*, performance-*)

/* Wandelt eine textuelle Ip-Adresse in ein USINT-Array */
unsigned short BrbIpToNumericalArray(plcstring* pIp, unsigned long pUsintArray)
{
	// Prüfung der Parameter
	if(pIp == 0)
	{
		return eBRB_ERR_NULL_POINTER;
	}
	if(pUsintArray == 0)
	{
		return eBRB_ERR_NULL_POINTER;
	}
	// Die einzelnen Segemente in ein String-Array kopieren
	STRING asIp[4][nBRB_IP_ADR_CHAR_MAX];
	BrbStringSplitEmpty(pIp, ".", (UDINT)&asIp, 3, sizeof(asIp[0]));
	// Die einzelnen Segemente in USINT wandeln
	UINT nIndex = 0;
	for(nIndex=0; nIndex<=3; nIndex++)
	{
		*(((USINT*)pUsintArray)+nIndex) = (USINT)brsatoi((UDINT)&asIp[nIndex]);
	}
	return eBRB_ERR_OK;
}

// NOLINTEND(readability-*, bugprone-easily-swappable-parameters, clang-diagnostic-invalid-utf8, clang-diagnostic-invalid-source-encoding, clang-diagnostic-pointer-arith, clang-diagnostic-strict-prototypes, hicpp-uppercase-literal-suffix, cppcoreguidelines-*, performance-*)
```

#### BrbCheckIpAddress.c - Prüft eine Ip-Adresse und berichtigt sie gegebenenfalls
```c
/********************************************************************
 * COPYRIGHT -- Bernecker + Rainer
 ********************************************************************
 * Library: BrbLib
 * File: BrbCheckIpAddress.c
 * Author: niedermeierr
 * Created: November 25, 2014
 ********************************************************************
 * Implementation of library BrbLib
 ********************************************************************/

#include <bur/plctypes.h>
#ifdef __cplusplus
	extern "C"
	{
#endif

#include "BrbLib.h"
#include <string.h>

#ifdef __cplusplus
	};
#endif

// NOLINTBEGIN(readability-*, bugprone-easily-swappable-parameters, clang-diagnostic-invalid-utf8, clang-diagnostic-invalid-source-encoding, clang-diagnostic-pointer-arith, clang-diagnostic-strict-prototypes, hicpp-uppercase-literal-suffix, cppcoreguidelines-*, performance-*)

/* Prüft eine Ip-Adresse und berichtigt sie gegebenenfalls */
plcbit BrbCheckIpAddress(plcstring* pIpAddress)
{
	// Eine Ip-Adresse darf keine Buchstaben enthalten.
	// Die einzelnen Segmente dürfen keine führenden Nullen haben, weil sie sonst vom Betriebssystem als Oktal-Zahl erkannt werden.
	BOOL bResult = 0;
	STRING sAdr[4][nBRB_IP_ADR_CHAR_MAX];
	BrbStringSplitEmpty(pIpAddress, ".", (UDINT)&sAdr, 3, sizeof(sAdr[0]));
	UINT nIndex = 0;
	for(nIndex=0; nIndex<=3; nIndex++)
	{
		UDINT nLen = strlen(sAdr[nIndex]);
		if(nLen == 0)
		{
			// Leerstring wird zu "0"
			strcpy(sAdr[nIndex], "0");
		}
		else
		{
			// Nummern-Prüfung
			DINT nNumber = brsatoi((UDINT)&sAdr[nIndex]);
			nNumber = ((nNumber > 255)? 255 : ((nNumber < 0)? 0 : nNumber)); // auf 0..255 limitieren
			brsitoa(nNumber, (UDINT)&sAdr[nIndex]);
		}
	}
	// NOLINTBEGIN(clang-analyzer-security.insecureAPI.strcpy)
	strcpy(pIpAddress, "");
	strcat(pIpAddress, sAdr[0]);
	strcat(pIpAddress, ".");
	strcat(pIpAddress, sAdr[1]);
	strcat(pIpAddress, ".");
	strcat(pIpAddress, sAdr[2]);
	strcat(pIpAddress, ".");
	strcat(pIpAddress, sAdr[3]);
	// NOLINTEND(clang-analyzer-security.insecureAPI.strcpy)
	return bResult;
}

// NOLINTEND(readability-*, bugprone-easily-swappable-parameters, clang-diagnostic-invalid-utf8, clang-diagnostic-invalid-source-encoding, clang-diagnostic-pointer-arith, clang-diagnostic-strict-prototypes, hicpp-uppercase-literal-suffix, cppcoreguidelines-*, performance-*)
```

#### BrbCheckSubnet.c - Prüft eine Subnet-Maske
```c
/********************************************************************
 * COPYRIGHT -- Bernecker + Rainer
 ********************************************************************
 * Library: BrbLib
 * File: BrbCheckSubnet.c
 * Author: niedermeierr
 * Created: July 05, 2022
 ********************************************************************
 * Implementation of library BrbLib
 ********************************************************************/

#include <bur/plctypes.h>
#ifdef __cplusplus
	extern "C"
	{
#endif

#include "BrbLib.h"
#include <string.h>

#ifdef __cplusplus
	};
#endif

// NOLINTBEGIN(readability-*, bugprone-easily-swappable-parameters, clang-diagnostic-invalid-utf8, clang-diagnostic-invalid-source-encoding, clang-diagnostic-pointer-arith, clang-diagnostic-strict-prototypes, hicpp-uppercase-literal-suffix, cppcoreguidelines-*, performance-*)

/* Prüft eine Subnet-Angabe auf Gültigkeit */
plcbit BrbCheckSubnet(plcstring* pSubnet)
{
	BOOL bResult = 1;
	// Subnet in numerisches Array wandeln
	USINT anSubnet[4];	BrbIpToNumericalArray(pSubnet, (UDINT)&anSubnet);
	// Sobald eine Null im Bitmuster gesetzt ist, dürfen nur noch Nullen folgen
	UINT nIndex = 0;
	BOOL bFollowingBitsMustBeZero = 0;
	for(nIndex=0; nIndex<=3; nIndex++)
	{
		// Es dürfen nur bestimmte Bitmuster in einem Segment gesetzt sein (nur führende Einsen)
		// NOLINTBEGIN(bugprone-branch-clone)
		if(bFollowingBitsMustBeZero && anSubnet[nIndex] != 0)
		{
			// Keine führende 1
			bResult = 0;
			break;
		}
		else if(anSubnet[nIndex] == 255)
		{
			// Alle Bits des Netzwerk-Anteils gesetzt -> Passt
		}
		else if(anSubnet[nIndex] == 0
		|| anSubnet[nIndex] == 128	// #1000 0000
		|| anSubnet[nIndex] == 192	// #1100 0000
		|| anSubnet[nIndex] == 224	// #1110 0000
		|| anSubnet[nIndex] == 240	// #1111 0000
		|| anSubnet[nIndex] == 248	// #1111 1000
		|| anSubnet[nIndex] == 252	// #1111 1100
		|| anSubnet[nIndex] == 254	// #1111 1110
		)
		{
			// Nur führende Einsen -> Nachfolgende Segmente dürfen kein Bit gesetzt haben
			bFollowingBitsMustBeZero = 1;
		}
		else
		{
			// Keine führende 1
			bResult = 0;
			break;
		}
		// NOLINTEND(bugprone-branch-clone)
	}
	// Zusätzliche Prüfungen
	UDINT* pSubnetUdint = (UDINT*)&anSubnet; // NOLINT(clang-diagnostic-cast-align)
	if(*pSubnetUdint == 0)
	{
		// Nur Nullen sind nicht erlaubt
		bResult = 0;
	}
	if(*pSubnetUdint == nBRB_UDINT_MAX)
	{
		// Nur Einsen sind nicht erlaubt
		bResult = 0;
	}
	return bResult;
}

// NOLINTEND(readability-*, bugprone-easily-swappable-parameters, clang-diagnostic-invalid-utf8, clang-diagnostic-invalid-source-encoding, clang-diagnostic-pointer-arith, clang-diagnostic-strict-prototypes, hicpp-uppercase-literal-suffix, cppcoreguidelines-*, performance-*)
```

#### BrbGetIpAddressType.c - Gibt den Typ einer Ip-Adresse zurück
```c
/********************************************************************
 * COPYRIGHT -- Bernecker + Rainer
 ********************************************************************
 * Library: BrbLib
 * File: BrbGetIpAddressType.c
 * Author: niedermeierr
 * Created: July 05, 2022
 ********************************************************************
 * Implementation of library BrbLib
 ********************************************************************/

#include <bur/plctypes.h>
#ifdef __cplusplus
	extern "C"
	{
#endif

#include "BrbLib.h"
#include <string.h>

#ifdef __cplusplus
	};
#endif

// NOLINTBEGIN(readability-*, bugprone-easily-swappable-parameters, clang-diagnostic-invalid-utf8, clang-diagnostic-invalid-source-encoding, clang-diagnostic-pointer-arith, clang-diagnostic-strict-prototypes, hicpp-uppercase-literal-suffix, cppcoreguidelines-*, performance-*)

/* Gibt den Typen einer Ip-Adresse zurück (Netzwerk-oder Broadcast-Adresse) */
enum BrbIpAdrType_ENUM BrbGetIpAddressType(plcstring* pIp, plcstring* pSubnet)
{
	BrbIpAdrType_ENUM eResult = eBRB_IP_ADR_TYPE_UNKNOWN;
	// Ip und Subnet in numerische Arrays wandeln
	USINT anIp[4];			BrbIpToNumericalArray(pIp, (UDINT)&anIp);
	USINT anSubnet[4];	BrbIpToNumericalArray(pSubnet, (UDINT)&anSubnet);
	USINT anSubnetComplement[4];
	USINT anNetworkIp[4];
	USINT anBroadcastIp[4];
	UINT nIndex = 0;
	for(nIndex=0; nIndex<=3; nIndex++)
	{
		// Komplement des Subnets bilden (Bits umkehren), um so den Host-Anteil zu bekommen
		anSubnetComplement[nIndex] = ~anSubnet[nIndex];
		// Netzwerk-Adresse aufgrund des Subnets ermitteln (kleinste Adresse des Host-Bereichs)
		anNetworkIp[nIndex] = (anIp[nIndex] & anSubnet[nIndex]);
		// Broadcast-Adresse aufgrund des Subnets ermitteln (größte Adresse des Host-Bereichs)
		anBroadcastIp[nIndex] = (anIp[nIndex] & anSubnet[nIndex]) | anSubnetComplement[nIndex]; // NOLINT(hicpp-signed-bitwise)
	}
	// Vergleich mit den ermittelten Adressen
	UDINT* pIpUdint = (UDINT*)&anIp; // NOLINT(clang-diagnostic-cast-align)
	UDINT* pNetworkIpUdint = (UDINT*)&anNetworkIp; // NOLINT(clang-diagnostic-cast-align)
	UDINT* pBroadcastIpUdint = (UDINT*)&anBroadcastIp; // NOLINT(clang-diagnostic-cast-align)
	// Da auf direkte Gleichheit geprüft werden muss, können die 4 Byte-Segmente jeweils vereinfacht als UDINT (ebenfalls 4 Byte) verglichen werden
	// NOLINTBEGIN(bugprone-branch-clone)
	if(*pIpUdint == 0)
	{
		eResult = eBRB_IP_ADR_TYPE_UNKNOWN;
	}
	else if(*pIpUdint == nBRB_UDINT_MAX)
	{
		eResult = eBRB_IP_ADR_TYPE_UNKNOWN;
	}
	else if(*pIpUdint == *pNetworkIpUdint)
	{
		eResult = eBRB_IP_ADR_TYPE_NETWORK;
	}
	else if(*pIpUdint == *pBroadcastIpUdint)
	{
		eResult = eBRB_IP_ADR_TYPE_BROADCAST;
	}
	else
	{
		eResult = eBRB_IP_ADR_TYPE_HOST;
	}
	// NOLINTEND(bugprone-branch-clone)
	return eResult;
}

// NOLINTEND(readability-*, bugprone-easily-swappable-parameters, clang-diagnostic-invalid-utf8, clang-diagnostic-invalid-source-encoding, clang-diagnostic-pointer-arith, clang-diagnostic-strict-prototypes, hicpp-uppercase-literal-suffix, cppcoreguidelines-*, performance-*)
```

#### BrbCheckIpEqualSubnet.c - Prüft, ob sich zwei Ip-Adressen im selben Subnet befinden
```c
/********************************************************************
 * COPYRIGHT -- Bernecker + Rainer
 ********************************************************************
 * Library: BrbLib
 * File: BrbCheckIpEqualSubnet.c
 * Author: niedermeierr
 * Created: July 05, 2022
 ********************************************************************
 * Implementation of library BrbLib
 ********************************************************************/

#include <bur/plctypes.h>
#ifdef __cplusplus
	extern "C"
	{
#endif

#include "BrbLib.h"
#include <string.h>

#ifdef __cplusplus
	};
#endif

// NOLINTBEGIN(readability-*, bugprone-easily-swappable-parameters, clang-diagnostic-invalid-utf8, clang-diagnostic-invalid-source-encoding, clang-diagnostic-pointer-arith, clang-diagnostic-strict-prototypes, hicpp-uppercase-literal-suffix, cppcoreguidelines-*, performance-*)

/* Prüft, ob zwei Ip-Adressen im selben Subnet sind */
plcbit BrbCheckIpEqualSubnet(plcstring* pIp1, plcstring* pSubnet1, plcstring* pIp2, plcstring* pSubnet2)
{
	BOOL bResult = 1;
	// Ip's und Subnets in numerische Arrays wandeln
	USINT anIp1[4];			BrbIpToNumericalArray(pIp1, (UDINT)&anIp1);
	USINT anSubnet1[4];	BrbIpToNumericalArray(pSubnet1, (UDINT)&anSubnet1);
	USINT anIp2[4];			BrbIpToNumericalArray(pIp2, (UDINT)&anIp2);
	USINT anSubnet2[4];	BrbIpToNumericalArray(pSubnet2, (UDINT)&anSubnet2);
	// Vergleich der Netz-Anteile (durch Verundung mit dem Subnet wird der Host-Anteil elimniert)
	UINT nIndex = 0;
	for(nIndex=0; nIndex<=3; nIndex++)
	{
		// Subnet verodern (das Subnet gibt den Netz-Anteil an, somit wird der gemeinsame Netz-Anteil zum Vergleich verwendet)
		USINT nSubnet = anSubnet1[nIndex] | anSubnet2[nIndex];
		// Vergleich
		USINT nIp1 = anIp1[nIndex] & nSubnet;
		USINT nIp2 = anIp2[nIndex] & nSubnet;
		if(nIp1 != nIp2)
		{
			bResult = 0;
			break;
		}
	}
	return bResult;
}

// NOLINTEND(readability-*, bugprone-easily-swappable-parameters, clang-diagnostic-invalid-utf8, clang-diagnostic-invalid-source-encoding, clang-diagnostic-pointer-arith, clang-diagnostic-strict-prototypes, hicpp-uppercase-literal-suffix, cppcoreguidelines-*, performance-*)
```

#### Package Logical/Libraries/BrbLib/Additional - Erzeugung von Zufallszahlen

#### BrbDebounceInput.c - Entprellt einen Eingang
```c
/********************************************************************
 * COPYRIGHT -- Bernecker + Rainer
 ********************************************************************
 * Library: BrbLib
 * File: BrbDebounceInput.c
 * Author: niedermeierr
 * Created: April 15, 2015
 ********************************************************************
 * Implementation of library BrbLib
 ********************************************************************/

#include <bur/plctypes.h>
#ifdef __cplusplus
	extern "C"
	{
#endif

#include "BrbLib.h"

#ifdef __cplusplus
	};
#endif

// NOLINTBEGIN(readability-*, bugprone-easily-swappable-parameters, clang-diagnostic-invalid-utf8, clang-diagnostic-invalid-source-encoding, clang-diagnostic-pointer-arith, clang-diagnostic-strict-prototypes, hicpp-uppercase-literal-suffix, cppcoreguidelines-*, performance-*)

/* Entprellt einen Eingang */
void BrbDebounceInput(struct BrbDebounceInput* inst)
{
	inst->bOutput = 0;
	inst->fbDebounce.PT = (TIME)inst->nDebounceTime;
	TON(&inst->fbDebounce);
	if(inst->fbDebounce.Q == 1)
	{
		inst->fbDebounce.IN = 0;
		TON(&inst->fbDebounce);
	}
	if(inst->bInput == 1 && inst->fbDebounce.IN == 0)
	{
		inst->bOutput = 1;
		inst->fbDebounce.IN = 1;
		TON(&inst->fbDebounce);
	}
}

// NOLINTEND(readability-*, bugprone-easily-swappable-parameters, clang-diagnostic-invalid-utf8, clang-diagnostic-invalid-source-encoding, clang-diagnostic-pointer-arith, clang-diagnostic-strict-prototypes, hicpp-uppercase-literal-suffix, cppcoreguidelines-*, performance-*)
```

#### BrbGetStructMemberOffset.c - Gibt den Offset eines Struktur-Members zurück
```c
/********************************************************************
 * COPYRIGHT -- Bernecker + Rainer
 ********************************************************************
 * Library: BrbLib
 * File: BrbGetStructMemberOffset.c
 * Author: niedermeierr
 * Created: December 21, 2015
 ********************************************************************
 * Implementation of library BrbLib
 ********************************************************************/

#include <bur/plctypes.h>
#ifdef __cplusplus
	extern "C"
	{
#endif

#include "BrbLib.h"
#include <string.h>

#ifdef __cplusplus
	};
#endif

// NOLINTBEGIN(readability-*, bugprone-easily-swappable-parameters, clang-diagnostic-invalid-utf8, clang-diagnostic-invalid-source-encoding, clang-diagnostic-pointer-arith, clang-diagnostic-strict-prototypes, hicpp-uppercase-literal-suffix, cppcoreguidelines-*, performance-*)

/* Gibt den Offset eines Struktur-Members zurück */
unsigned short BrbGetStructMemberOffset(plcstring* pStructName, plcstring* pMemberName, unsigned long* pOffset)
{
	UINT nStatus = 0;
	*pOffset = 0;
	// Adresse der Struktur-Instanz ermitteln
	UDINT nAddressStruct = 0;
	UDINT nLen = 0;
	nStatus = PV_xgetadr((STRING*)pStructName, (UDINT*)&nAddressStruct, (UDINT*)&nLen);
	if(nStatus == 0)
	{
		// Adresse der Struktur-Member ermitteln
		UDINT nAddressMember = 0;
		STRING sMember[nBRB_PVNAME_CHAR_MAX];
		BrbStringCopy(sMember, pStructName, sizeof(sMember));
		BrbStringCat(sMember, ".", sizeof(sMember));
		BrbStringCat(sMember, pMemberName, sizeof(sMember));
		nStatus = PV_xgetadr((STRING*)&sMember, (UDINT*)&nAddressMember, (UDINT*)&nLen);
		if(nStatus == 0)
		{
			// Differenz ergibt Offset
			*pOffset = nAddressMember - nAddressStruct;
		}
	}
	return nStatus;
}

// NOLINTEND(readability-*, bugprone-easily-swappable-parameters, clang-diagnostic-invalid-utf8, clang-diagnostic-invalid-source-encoding, clang-diagnostic-pointer-arith, clang-diagnostic-strict-prototypes, hicpp-uppercase-literal-suffix, cppcoreguidelines-*, performance-*)
```

#### BrbGetCompilerVersion.c - Gibt die Version des Compilers zurück
```c
/********************************************************************
 * COPYRIGHT -- Bernecker + Rainer
 ********************************************************************
 * Library: BrbLib
 * File: BrbGetCompilerVersion.c
 * Author: niedermeierr
 * Created: October 24, 2019
 ********************************************************************
 * Implementation of library BrbLib
 ********************************************************************/

#include <bur/plctypes.h>
#ifdef __cplusplus
	extern "C"
	{
#endif

#include "BrbLib.h"
#include <string.h>

#ifdef __cplusplus
	};
#endif

// NOLINTBEGIN(readability-*, bugprone-easily-swappable-parameters, clang-diagnostic-invalid-utf8, clang-diagnostic-invalid-source-encoding, clang-diagnostic-pointer-arith, clang-diagnostic-strict-prototypes, hicpp-uppercase-literal-suffix, cppcoreguidelines-*, performance-*)

/* Gibt die Version des verwendeten GCC-Compilers zurück */
unsigned short BrbGetCompilerVersion(struct BrbCompilerVersion_TYP* pCompilerVersion)
{
	UINT nResult = 0;
	STRING sItoA[20];
	pCompilerVersion->bValid = 0;
	pCompilerVersion->nMajor = 0;
	pCompilerVersion->nMinor = 0;
	pCompilerVersion->nPatch = 0;
	pCompilerVersion->nTotal = 0;
	memset(&pCompilerVersion->sText, 0, sizeof(pCompilerVersion->sText));

	#ifdef __GNUC__
		pCompilerVersion->nMajor = __GNUC__;
		nResult += 4;
	#endif
	pCompilerVersion->nTotal += ((DINT)pCompilerVersion->nMajor * 10000);
	brsitoa((DINT)pCompilerVersion->nMajor, (UDINT)&sItoA);
	BrbStringCopy((STRING*)&pCompilerVersion->sText, sItoA, sizeof(pCompilerVersion->sText));
	BrbStringCat((STRING*)&pCompilerVersion->sText, ".", sizeof(pCompilerVersion->sText));

	#ifdef __GNUC_MINOR__
		pCompilerVersion->nMinor = __GNUC_MINOR__;
		nResult += 2;
	#endif
	pCompilerVersion->nTotal += ((DINT)pCompilerVersion->nMinor * 100);
	brsitoa((DINT)pCompilerVersion->nMinor, (UDINT)&sItoA);
	BrbStringCat((STRING*)&pCompilerVersion->sText, sItoA, sizeof(pCompilerVersion->sText));
	BrbStringCat((STRING*)&pCompilerVersion->sText, ".", sizeof(pCompilerVersion->sText));

	#ifdef __GNUC_PATCHLEVEL__
		pCompilerVersion->nPatch = __GNUC_PATCHLEVEL__;
		nResult += 1;
	#endif
	pCompilerVersion->nTotal += (DINT)pCompilerVersion->nPatch;
	brsitoa((DINT)pCompilerVersion->nPatch, (UDINT)&sItoA);
	BrbStringCat((STRING*)&pCompilerVersion->sText, sItoA, sizeof(pCompilerVersion->sText));

	if(nResult >= 7)
	{
		pCompilerVersion->bValid = 1;
	}
	return nResult;
}

// NOLINTEND(readability-*, bugprone-easily-swappable-parameters, clang-diagnostic-invalid-utf8, clang-diagnostic-invalid-source-encoding, clang-diagnostic-pointer-arith, clang-diagnostic-strict-prototypes, hicpp-uppercase-literal-suffix, cppcoreguidelines-*, performance-*)
```

### Library Logical/Libraries/BrbLibUa (ANSIC, version 1.03.0) - Helpful OpcUa functions
Depends on: AsOpcUac, AsOpcUas, BrbLib, DataObj, FileIO

#### License.txt
```
MIT License

Copyright (c) [2021] [Rainer Niedermeier]

Permission is hereby granted, free of charge, to any person obtaining a copy
of this software and associated documentation files (the "Software"), to deal
in the Software without restriction, including without limitation the rights
to use, copy, modify, merge, publish, distribute, sublicense, and/or sell
copies of the Software, and to permit persons to whom the Software is
furnished to do so, subject to the following conditions:

The above copyright notice and this permission notice shall be included in all
copies or substantial portions of the Software.

THE SOFTWARE IS PROVIDED "AS IS", WITHOUT WARRANTY OF ANY KIND, EXPRESS OR
IMPLIED, INCLUDING BUT NOT LIMITED TO THE WARRANTIES OF MERCHANTABILITY,
FITNESS FOR A PARTICULAR PURPOSE AND NONINFRINGEMENT. IN NO EVENT SHALL THE
AUTHORS OR COPYRIGHT HOLDERS BE LIABLE FOR ANY CLAIM, DAMAGES OR OTHER
LIABILITY, WHETHER IN AN ACTION OF CONTRACT, TORT OR OTHERWISE, ARISING FROM,
OUT OF OR IN CONNECTION WITH THE SOFTWARE OR THE USE OR OTHER DEALINGS IN THE
SOFTWARE.
```

#### BrbLibUa.fun - Exported functions and function blocks
```iecst
(*General - Status*)

FUNCTION BrbUaGetStatusCodeText : DWORD (*Gibt den symbolischen Text für einen Ua-Status-Code zurück*) (*$GROUP=User,$CAT=User,$GROUPICON=User.png,$CATICON=User.png*)
	VAR_INPUT
		nStatusCode : UDINT; (*Status-Code*)
		pStatusText : STRING[0]; (*Zeiger auf Text*)
		nStatusTextSize : UDINT; (*Größe des Textes*)
	END_VAR
END_FUNCTION
(*General - Nodes*)

FUNCTION BrbUaSetNodeId : DWORD (*Besetzt eine NodeId*) (*$GROUP=User,$CAT=User,$GROUPICON=User.png,$CATICON=User.png*)
	VAR_INPUT
		pNodeId : UANodeID; (*Zeiger auf die NodeId*)
		sIdentifier : STRING[0]; (*Knoten-Name*)
		nNamespaceIndex : UINT; (*Namensraum-Index*)
	END_VAR
END_FUNCTION

FUNCTION BrbUaSetNodeIdNum : DWORD (*Besetzt eine numerische NodeId*) (*$GROUP=User,$CAT=User,$GROUPICON=User.png,$CATICON=User.png*)
	VAR_INPUT
		pNodeId : UANodeID; (*Zeiger auf die NodeId*)
		nIdentifier : UDINT; (*Knoten-Nummer*)
		nNamespaceIndex : UINT; (*Namensraum-Index*)
	END_VAR
END_FUNCTION

FUNCTION BrbUaGetRandomNodeId : DWORD (*Erzeugt eine zufällige NodeId*) (*$GROUP=User,$CAT=User,$GROUPICON=User.png,$CATICON=User.png*)
	VAR_INPUT
		pNodeId : UANodeID; (*Zeiger auf die NodeId*)
		eIdentifierType : UAIdentifierType; (*UAIdentifierType_String, Numeric, GUID oder Opaque*)
	END_VAR
END_FUNCTION

FUNCTION BrbUaAreNodeIdsEqual : BOOL (*Gibt zurück, ob zwei NodeIds gleich sind*) (*$GROUP=User,$CAT=User,$GROUPICON=User.png,$CATICON=User.png*)
	VAR_INPUT
		pNodeId1 : UANodeID; (*Zeiger auf die erste NodeId*)
		pNodeId2 : UANodeID; (*Zeiger auf die zweite NodeId*)
	END_VAR
END_FUNCTION

FUNCTION BrbUaAddNodeIdText : DWORD (*Hängt den Text einer NodeId an*) (*$GROUP=User,$CAT=User,$GROUPICON=User.png,$CATICON=User.png*)
	VAR_INPUT
		pNodeId : UANodeID; (*Zeiger auf Quelle*)
		pText : STRING[0]; (*Zeiger auf Text*)
		nTextSize : UDINT; (*Größe des Textes*)
	END_VAR
END_FUNCTION
(*General - Attributes*)

FUNCTION BrbUaGetAttributeIdDatatype : UAVariantType (*Gibt den OpcUa-Datentyp für ein Attribut zurück*) (*$GROUP=User,$CAT=User,$GROUPICON=User.png,$CATICON=User.png*)
	VAR_INPUT
		eAttributeId : UAAttributeId; (*Attribut*)
	END_VAR
END_FUNCTION

FUNCTION BrbUaGetAttributeList : DWORD (*Gibt eine Liste mit Attribut-Texten zurück*) (*$GROUP=User,$CAT=User,$GROUPICON=User.png,$CATICON=User.png*)
	VAR_INPUT
		pNodeInfo : UANodeInfo; (*Zeiger auf die NodeInfo*)
		pAttributes : BrbUaNodeInfoAttributes_TYP; (*Zeiger auf die Liste der Attrbute*)
	END_VAR
END_FUNCTION

FUNCTION BrbUaAddBooleanText : DWORD (*Hängt den Text eines boolschen Werts an*) (*$GROUP=User,$CAT=User,$GROUPICON=User.png,$CATICON=User.png*)
	VAR_INPUT
		bBoolean : BOOL; (*Quelle*)
		pText : STRING[0]; (*Zeiger auf Text*)
		nTextSize : UDINT; (*Größe des Textes*)
	END_VAR
END_FUNCTION

FUNCTION BrbUaAddNodeClassText : DWORD (*Hängt den Text einer NodeClass an*) (*$GROUP=User,$CAT=User,$GROUPICON=User.png,$CATICON=User.png*)
	VAR_INPUT
		eNodeClass : UANodeClass; (*Quelle*)
		pText : STRING[0]; (*Zeiger auf Text*)
		nTextSize : UDINT; (*Größe des Textes*)
	END_VAR
END_FUNCTION

FUNCTION BrbUaAddDatatypeIdText : DWORD (*Hängt den Text zu einem Datentyp-Identifier an*)
	VAR_INPUT
		nDatatypeId : UDINT; (*Quelle*)
		pText : STRING[0]; (*Zeiger auf Text*)
		nTextSize : UDINT; (*Größe des Textes*)
	END_VAR
END_FUNCTION

FUNCTION BrbUaAddArrayDimensionText : DWORD (*Hängt den Text für eine ArrayDimension an*) (*$GROUP=User,$CAT=User,$GROUPICON=User.png,$CATICON=User.png*)
	VAR_INPUT
		pArrayDimension : REFERENCE TO UDINT; (*Zeiger auf Quelle*)
		nValueRank : DINT; (*Anzahl der Dimensionen*)
		pText : STRING[0]; (*Zeiger auf Text*)
		nTextSize : UDINT; (*Größe des Textes*)
	END_VAR
END_FUNCTION

FUNCTION BrbUaAddAccessLevelText : DWORD (*Hängt den Text eines AccessLevels an*) (*$GROUP=User,$CAT=User,$GROUPICON=User.png,$CATICON=User.png*)
	VAR_INPUT
		nAccessLevel : BYTE; (*Quelle*)
		pText : STRING[0]; (*Zeiger auf Text*)
		nTextSize : UDINT; (*Größe des Textes*)
	END_VAR
END_FUNCTION

FUNCTION BrbUaAddEventNotifierText : DWORD (*Hängt den Text eines EventNotifiers an*) (*$GROUP=User,$CAT=User,$GROUPICON=User.png,$CATICON=User.png*)
	VAR_INPUT
		nEventNotifier : BYTE; (*Quelle*)
		pText : STRING[0]; (*Zeiger auf Text*)
		nTextSize : UDINT; (*Größe des Textes*)
	END_VAR
END_FUNCTION
(*General - VariantValues*)

FUNCTION BrbUaClearVariantValue : DWORD (*Löscht den Inhalt eines OpcUa-Values, aber nicht die Datentyp-Angabe*) (*$GROUP=User,$CAT=User,$GROUPICON=User.png,$CATICON=User.png*)
	VAR_INPUT
		pUaVariantData : UAVariantData; (*Zeiger auf Variant*)
	END_VAR
END_FUNCTION

FUNCTION BrbUaConvVariantValueFromString : DWORD (*Wandelt einen OpcUa-Value in einen Text*) (*$GROUP=User,$CAT=User,$GROUPICON=User.png,$CATICON=User.png*)
	VAR_INPUT
		pUaVariantData : UAVariantData; (*Zeiger auf Variant*)
		pValueText : STRING[0]; (*Zeiger auf Text*)
	END_VAR
END_FUNCTION

FUNCTION BrbUaConvVariantValueToString : DWORD (*Wandelt einen Text in einen OpcUa-Value*) (*$GROUP=User,$CAT=User,$GROUPICON=User.png,$CATICON=User.png*)
	VAR_INPUT
		pUaVariantData : UAVariantData; (*Zeiger auf Variant#*)
		pValueText : STRING[0]; (*Zeiger auf Text*)
		nValueTextSize : UDINT; (*Größe des Textes*)
	END_VAR
END_FUNCTION

FUNCTION BrbUaAddVariantValueSubName : DWORD (*Hängt den Element-Namen eines OpcUa-Values anhand des Datentypen an einen Text an*) (*$GROUP=User,$CAT=User,$GROUPICON=User.png,$CATICON=User.png*)
	VAR_INPUT
		eVariantType : UAVariantType; (*Datentyp*)
		pText : STRING[0]; (*Zeiger auf Text*)
		nTextSize : UDINT; (*Größe des Textes*)
	END_VAR
END_FUNCTION
(*General - ByteStrings*)

FUNCTION BrbUaIncByteString : DWORD (*Inkrementiert einen ByteString*) (*$GROUP=User,$CAT=User,$GROUPICON=User.png,$CATICON=User.png*)
	VAR_INPUT
		pData : REFERENCE TO USINT; (*Zeiger auf das Daten-Array des ByteStrings*)
		nLength : DINT; (*Länge des Daten-Arrays*)
	END_VAR
END_FUNCTION

FUNCTION BrbUaGetRandomByteString : DWORD (*Erzeugt einen zufälligen ByteString*) (*$GROUP=User,$CAT=User,$GROUPICON=User.png,$CATICON=User.png*)
	VAR_INPUT
		pData : REFERENCE TO USINT; (*Zeiger auf das Daten-Array des ByteStrings*)
		nLength : DINT; (*Länge des Daten-Arrays*)
	END_VAR
END_FUNCTION
(*General - Images*)

{REDUND_UNREPLICABLE} FUNCTION_BLOCK BrbUaLoadImage (*Lädt ein Image*) (*$GROUP=User,$CAT=User,$GROUPICON=User.png,$CATICON=User.png*)
	VAR_INPUT
		pDevice : REFERENCE TO STRING[0]; (*Zeiger auf den Laufwerks-Namen*)
		pFile : REFERENCE TO STRING[0]; (*Zeiger auf den Datei-Namen*)
		pImageData : REFERENCE TO USINT; (*Zeiger auf die Image-Daten*)
		nImageDataSize : {REDUND_UNREPLICABLE} UDINT; (*Größe der Image-Daten*)
		pImageLength : REFERENCE TO DINT; (*Zeiger auf die Image-Länge*)
	END_VAR
	VAR_OUTPUT
		nStatus : {REDUND_UNREPLICABLE} UINT; (*Fub-Status*)
	END_VAR
	VAR
		eStep : {REDUND_UNREPLICABLE} DINT; (*Step-Nummer für die interne Schrittkette*)
		fbBrbLoadFileBin : {REDUND_UNREPLICABLE} BrbLoadFileBin; (*Interner Fub*)
	END_VAR
END_FUNCTION_BLOCK
(*General - LocalizedTexts*)

FUNCTION BrbUaSetLocalizedText : DWORD (*Besetzt einen LocalizedText*) (*$GROUP=User,$CAT=User,$GROUPICON=User.png,$CATICON=User.png*)
	VAR_INPUT
		pLocalizedText : REFERENCE TO BrUaLocalizedText; (*Zeiger auf den LocalizedText*)
		pLocale : STRING[0]; (*Locale-Angabe*)
		pText : STRING[0]; (*Text-Angabe*)
	END_VAR
END_FUNCTION

FUNCTION BrbUaGetRandomLocalizedText : DWORD (*Erzeugt einen zufälligen LocalizedText*) (*$GROUP=User,$CAT=User,$GROUPICON=User.png,$CATICON=User.png*)
	VAR_INPUT
		pLocalizedText : REFERENCE TO BrUaLocalizedText; (*Zeiger auf den LocalizedText*)
		nLength : UINT; (*Zu erzeugende Länge des Textes*)
	END_VAR
END_FUNCTION

FUNCTION BrbUaAddLocalizedTextText : DWORD (*Hängt den Text eines LocalizedText an*) (*$GROUP=User,$CAT=User,$GROUPICON=User.png,$CATICON=User.png*)
	VAR_INPUT
		pLocalizedText : REFERENCE TO BrUaLocalizedText; (*Zeiger auf den LocalizedText*)
		pText : STRING[0]; (*Zeiger auf Text*)
		nTextSize : UDINT; (*Größe des Textes*)
	END_VAR
END_FUNCTION
(*General - QualifiedNames*)

FUNCTION BrbUaSetQualifedName : DWORD (*Besetzt einen QualifiedName*) (*$GROUP=User,$CAT=User,$GROUPICON=User.png,$CATICON=User.png*)
	VAR_INPUT
		pQualifiedName : REFERENCE TO BrUaQualifiedName; (*Zeiger auf den QualifiedName*)
		nNamespaceIndex : UINT; (*Namensraum-Index*)
		pName : STRING[0]; (*Zeiger auf den Namen*)
	END_VAR
END_FUNCTION

FUNCTION BrbUaGetRandomQualifiedName : DWORD (*Erzeugt einen zufälligen QualifiedName*) (*$GROUP=User,$CAT=User,$GROUPICON=User.png,$CATICON=User.png*)
	VAR_INPUT
		pQualifiedName : REFERENCE TO BrUaQualifiedName; (*Zeiger auf den QualifiedName*)
		nLength : UINT; (*Zu erzeugende Länge des Namens*)
	END_VAR
END_FUNCTION
(*General - TimeAndDate*)

FUNCTION BrbUaDtStructToUaSrvDateTime : UINT (*Wandelt eine DtStruct-Zeit in eine UaSrvDateTime-Zeit*) (*$GROUP=User,$CAT=User,$GROUPICON=User.png,$CATICON=User.png*)
	VAR_INPUT
		pUaSrvDateTime : UaSrv_DateTimeType; (*Zeiger auf eine Struktur "UaSrv_DateTimeType"*)
		pDtStruct : DTStructure; (*Zeiger auf eine Struktur "DTStructure"*)
		nNanoSeconds : UINT; (*Anzahl der Nano-Sekunden (0..999)*)
	END_VAR
END_FUNCTION

FUNCTION BrbUaSrvDateTimeToDtStruct : UINT (*Wandelt eine UaSrvDateTime-Zeit in eine DtStruct-Zeit*) (*$GROUP=User,$CAT=User,$GROUPICON=User.png,$CATICON=User.png*)
	VAR_INPUT
		pDtStruct : DTStructure; (*Zeiger auf eine Struktur "DTStructure"*)
		pUaSrvDateTime : UaSrv_DateTimeType; (*Zeiger auf eine Struktur "UaSrv_DateTimeType"*)
	END_VAR
END_FUNCTION

FUNCTION BrbUaGetSrvTimeText : UINT (*Gibt den Text eines Server-Zeitstempels zurück*) (*$GROUP=User,$CAT=User,$GROUPICON=User.png,$CATICON=User.png*)
	VAR_INPUT
		pSrvTime : UaSrv_DateTimeType; (*Zeiger auf eine Zeit-Struktur*)
		pText : STRING[0]; (*Zeiger auf den String*)
		nTextSize : UDINT; (*Größe der String-Variablen*)
		nTimeOffset : INT; (*Lokaler Zeit-Offset in [min]*)
		pFormat : STRING[0]; (*Zeiger auf den Formatierungstext*)
	END_VAR
END_FUNCTION

FUNCTION BrbUaGetRandomTimeZone : DWORD (*Erzeugt eine zufällige TimeZone*) (*$GROUP=User,$CAT=User,$GROUPICON=User.png,$CATICON=User.png*)
	VAR_INPUT
		pTimeZone : REFERENCE TO BrUaTimeZoneDataType; (*Zeiger auf die TimeZone*)
	END_VAR
END_FUNCTION
(*General - Additional*)

FUNCTION BrbUaGetRandomGuidString : DWORD (*Erzeugt einen zufälligen GuidString im Format '01234567-0123-0123-0123-0123456789AB'*) (*$GROUP=User,$CAT=User,$GROUPICON=User.png,$CATICON=User.png*)
	VAR_INPUT
		pGuidString : REFERENCE TO BrUaGuidString; (*Zeiger auf den GuidString*)
		nGuidStringSize : UDINT; (*Größe des Textes*)
		bWithSeparator : BOOL; (*1=Mit Trennzeichen -*)
	END_VAR
END_FUNCTION

FUNCTION BrbUaGetRandomXmlElement : DWORD (*Erzeugt ein zufälliges XmlElement im Format '<Tag Attribute="X">Value</Tag>'*) (*$GROUP=User,$CAT=User,$GROUPICON=User.png,$CATICON=User.png*)
	VAR_INPUT
		pXmlElement : BrUaXmlElement; (*Zeiger auf das XmlElement*)
	END_VAR
END_FUNCTION
(*Client - Connection*)

FUNCTION BrbUaGetConnectionStatusText : DWORD (*Gibt einen Verbindungs-Status als Text zurück*) (*$GROUP=User,$CAT=User,$GROUPICON=User.png,$CATICON=User.png*)
	VAR_INPUT
		eConnectionStatus : UAConnectionStatus; (*Verbindungs-Status*)
		pStatusText : STRING[0]; (*Zeiger auf Text*)
		nStatusTextSize : UDINT; (*Größe des Textes*)
	END_VAR
END_FUNCTION
(*Client - RunClient*)

{REDUND_UNREPLICABLE} FUNCTION_BLOCK BrbUaRunClientInit (*Initialisiert eine Client-Instanz*) (*$GROUP=User,$CAT=User,$GROUPICON=User.png,$CATICON=User.png*)
	VAR_INPUT
		pRunClient : REFERENCE TO BrbUaRunClient_TYP; (*Zeiger auf die RunClient-Struktur*)
	END_VAR
	VAR_OUTPUT
		nStatus : {REDUND_UNREPLICABLE} UINT; (*Fub-Status*)
	END_VAR
	VAR
		eStep : {REDUND_UNREPLICABLE} DINT; (*Step-Nummer für die interne Schrittkette*)
		fbDatObjInfo : {REDUND_UNREPLICABLE} DatObjInfo; (*Interner FB*)
		fbDatObjRead : {REDUND_UNREPLICABLE} DatObjRead; (*Interner FB*)
		nAllocStatus : {REDUND_UNREPLICABLE} UINT; (*Interne Variable*)
		nNamespaceIndex : {REDUND_UNREPLICABLE} DINT; (*Interne Variable*)
		nNodeHandleIndex : {REDUND_UNREPLICABLE} DINT; (*Interne Variable*)
		nReadBlockIndex : {REDUND_UNREPLICABLE} DINT; (*Interne Variable*)
		nReadItemIndex : {REDUND_UNREPLICABLE} DINT; (*Interne Variable*)
		nWriteBlockIndex : {REDUND_UNREPLICABLE} DINT; (*Interne Variable*)
		nWriteItemIndex : {REDUND_UNREPLICABLE} DINT; (*Interne Variable*)
		nMethodIndex : {REDUND_UNREPLICABLE} DINT; (*Interne Variable*)
		nArgumentInputIndex : {REDUND_UNREPLICABLE} DINT; (*Interne Variable*)
		nArgumentOutputIndex : {REDUND_UNREPLICABLE} DINT; (*Interne Variable*)
		nSubscriptionIndex : {REDUND_UNREPLICABLE} DINT; (*Interne Variable*)
		nMonItemIndex : {REDUND_UNREPLICABLE} DINT; (*Interne Variable*)
		nEventItemIndex : {REDUND_UNREPLICABLE} DINT; (*Interne Variable*)
		nEventFieldIndex : {REDUND_UNREPLICABLE} DINT; (*Interne Variable*)
		nLoopIndex : {REDUND_UNREPLICABLE} UINT; (*Interne Variable*)
		sLine : {REDUND_UNREPLICABLE} STRING[1024]; (*Interne Variable*)
		nLineLen : {REDUND_UNREPLICABLE} UDINT; (*Interne Variable*)
		sValue : {REDUND_UNREPLICABLE} STRING[1024]; (*Interne Variable*)
		nValue : {REDUND_UNREPLICABLE} DINT; (*Interne Variable*)
		rValue : {REDUND_UNREPLICABLE} REAL; (*Interne Variable*)
		sVarName : {REDUND_UNREPLICABLE} STRING[nBRBUA_VARNAME_TEXT_CHAR_MAX]; (*Interne Variable*)
	END_VAR
END_FUNCTION_BLOCK

{REDUND_UNREPLICABLE} FUNCTION_BLOCK BrbUaRunClientCyclic (*Behandelt eine Client-Instanz*) (*$GROUP=User,$CAT=User,$GROUPICON=User.png,$CATICON=User.png*)
	VAR_INPUT
		pRunClient : REFERENCE TO BrbUaRunClient_TYP; (*Zeiger auf die RunClient-Struktur*)
	END_VAR
	VAR_OUTPUT
		nStatus : {REDUND_UNREPLICABLE} UINT; (*Fub-Status*)
	END_VAR
	VAR
		eStep : {REDUND_UNREPLICABLE} DINT; (*Step-Nummer für die interne Schrittkette*)
		fbUA_Connect : {REDUND_UNREPLICABLE} UA_Connect; (*Interner FB*)
		eCmdOld : {REDUND_UNREPLICABLE} BrbUaRcCommandos_ENUM; (*Interne Variable*)
		fbUA_GetNamespaceIndex : {REDUND_UNREPLICABLE} UA_GetNamespaceIndex; (*Interner FB*)
		nNamespaceIndex : {REDUND_UNREPLICABLE} DINT; (*Interne Variable*)
		fbUA_NodeGetHandleList : {REDUND_UNREPLICABLE} UA_NodeGetHandleList; (*Interner FB*)
		nNodeHandleIndex : {REDUND_UNREPLICABLE} DINT; (*Interne Variable*)
		nReadBlockIndex : {REDUND_UNREPLICABLE} DINT; (*Interne Variable*)
		nWriteBlockIndex : {REDUND_UNREPLICABLE} DINT; (*Interne Variable*)
		fbUA_MethodGetHandle : {REDUND_UNREPLICABLE} UA_MethodGetHandle; (*Interner FB*)
		nMethodIndex : {REDUND_UNREPLICABLE} DINT; (*Interne Variable*)
		fbUA_SubscriptionCreate : {REDUND_UNREPLICABLE} UA_SubscriptionCreate; (*Interner FB*)
		nSubscriptionIndex : {REDUND_UNREPLICABLE} DINT; (*Interne Variable*)
		fbUA_MonitoredItemAddList : {REDUND_UNREPLICABLE} UA_MonitoredItemAddList; (*Interner FB*)
		nMonItemIndex : {REDUND_UNREPLICABLE} DINT; (*Interne Variable*)
		nEventItemIndex : {REDUND_UNREPLICABLE} DINT; (*Interne Variable*)
		nEventFieldIndex : {REDUND_UNREPLICABLE} DINT; (*Interne Variable*)
		nLoopIndex : {REDUND_UNREPLICABLE} UINT; (*Interne Variable*)
		sVarName : {REDUND_UNREPLICABLE} STRING[nBRBUA_VARNAME_TEXT_CHAR_MAX]; (*Interne Variable*)
		fbUA_NodeGetHandle : {REDUND_UNREPLICABLE} UA_NodeGetHandle; (*Interner FB*)
		fbUA_EventItemAdd : {REDUND_UNREPLICABLE} UA_EventItemAdd; (*Interner FB*)
		fbUA_ConnectionGetStatus : {REDUND_UNREPLICABLE} UA_ConnectionGetStatus; (*Interner FB*)
		eClientStateOld : {REDUND_UNREPLICABLE} BrbUaRcClientStates_ENUM;
		bEventItemFound : {REDUND_UNREPLICABLE} BOOL; (*Interne Variable*)
		pEventItemReceived : REFERENCE TO BOOL; (*Interne Variable*)
		fbUA_EventItemOperate : {REDUND_UNREPLICABLE} UA_EventItemOperate; (*Interner FB*)
		fbUA_Disconnect : {REDUND_UNREPLICABLE} UA_Disconnect; (*Interner FB*)
	END_VAR
END_FUNCTION_BLOCK

{REDUND_UNREPLICABLE} FUNCTION_BLOCK BrbUaRunClientExit (*Exilisiert eine Client-Instanz*) (*$GROUP=User,$CAT=User,$GROUPICON=User.png,$CATICON=User.png*)
	VAR_INPUT
		pRunClient : REFERENCE TO BrbUaRunClient_TYP; (*Zeiger auf die RunClient-Struktur*)
	END_VAR
	VAR_OUTPUT
		nStatus : {REDUND_UNREPLICABLE} UINT; (*Fub-Status*)
	END_VAR
	VAR
		eStep : {REDUND_UNREPLICABLE} DINT; (*Step-Nummer für die interne Schrittkette*)
		fbUA_Disconnect : {REDUND_UNREPLICABLE} UA_Disconnect; (*Interner FB*)
		nReadBlockIndex : {REDUND_UNREPLICABLE} DINT; (*Interne Variable*)
		nWriteBlockIndex : {REDUND_UNREPLICABLE} DINT; (*Interne Variable*)
		nSubscriptionIndex : {REDUND_UNREPLICABLE} DINT; (*Interne Variable*)
		nEventItemIndex : {REDUND_UNREPLICABLE} DINT; (*Interne Variable*)
		nFreeStatus : {REDUND_UNREPLICABLE} UINT; (*Interne Variable*)
	END_VAR
END_FUNCTION_BLOCK

FUNCTION_BLOCK BrbUaRcReadBlock (*Liest eine ReadBlock vom Server*) (*$GROUP=User,$CAT=User,$GROUPICON=User.png,$CATICON=User.png*)
	VAR_INPUT
		pRunClient : REFERENCE TO BrbUaRunClient_TYP; (*Zeiger auf die RunClient-Struktur*)
		nReadBlockIndex : {REDUND_UNREPLICABLE} UINT; (*0-basierter Index des ReadBlocks*)
	END_VAR
	VAR_OUTPUT
		nStatus : {REDUND_UNREPLICABLE} UINT; (*Fub-Status*)
		nErrorId : {REDUND_UNREPLICABLE} DWORD; (*OpcUa-Fehler-Status*)
		sErrorId : {REDUND_UNREPLICABLE} STRING[nBRBUA_STATUS_TEXT_CHAR_MAX]; (*OpcUa-Fehler-Text*)
		nReadCount : UDINT; (*Anzahl der Reads*)
	END_VAR
	VAR
		eStep : {REDUND_UNREPLICABLE} DINT; (*Step-Nummer für die interne Schrittkette*)
		fbUaClt_ReadBulk : {REDUND_UNREPLICABLE} UaClt_ReadBulk; (*Interner FB*)
	END_VAR
END_FUNCTION_BLOCK

{REDUND_UNREPLICABLE} FUNCTION_BLOCK BrbUaRcWriteBlock (*Liest eine ReadBlock vom Server*) (*$GROUP=User,$CAT=User,$GROUPICON=User.png,$CATICON=User.png*)
	VAR_INPUT
		pRunClient : REFERENCE TO BrbUaRunClient_TYP; (*Zeiger auf die RunClient-Struktur*)
		nWriteBlockIndex : {REDUND_UNREPLICABLE} UINT; (*0-basierter Index des WriteBlocks*)
	END_VAR
	VAR_OUTPUT
		nStatus : {REDUND_UNREPLICABLE} UINT; (*Fub-Status*)
		nErrorId : {REDUND_UNREPLICABLE} DWORD; (*OpcUa-Fehler-Status*)
		sErrorId : {REDUND_UNREPLICABLE} STRING[nBRBUA_STATUS_TEXT_CHAR_MAX]; (*OpcUa-Fehler-Text*)
		nWriteCount : {REDUND_UNREPLICABLE} UDINT; (*Anzahl der Writes*)
	END_VAR
	VAR
		eStep : {REDUND_UNREPLICABLE} DINT; (*Step-Nummer für die interne Schrittkette*)
		fbUaClt_WriteBulk : {REDUND_UNREPLICABLE} UaClt_WriteBulk; (*Interner FB*)
	END_VAR
END_FUNCTION_BLOCK

{REDUND_UNREPLICABLE} FUNCTION_BLOCK BrbUaRcCallMethod (*Liest eine ReadBlock vom Server*) (*$GROUP=User,$CAT=User,$GROUPICON=User.png,$CATICON=User.png*)
	VAR_INPUT
		pRunClient : REFERENCE TO BrbUaRunClient_TYP; (*Zeiger auf die RunClient-Struktur*)
		nMethodIndex : {REDUND_UNREPLICABLE} UINT; (*0-basierter Index der Method*)
	END_VAR
	VAR_OUTPUT
		bInit : {REDUND_UNREPLICABLE} BOOL; (*Vor dem Call für einen Zyklus auf 1*)
		nStatus : {REDUND_UNREPLICABLE} UINT; (*Fub-Status*)
		nErrorId : {REDUND_UNREPLICABLE} DWORD; (*OpcUa-Fehler-Status*)
		sErrorId : {REDUND_UNREPLICABLE} STRING[nBRBUA_STATUS_TEXT_CHAR_MAX]; (*OpcUa-Fehler-Text*)
		nCallCount : {REDUND_UNREPLICABLE} UDINT; (*Anzahl der Calls*)
	END_VAR
	VAR
		nArgumentIndex : {REDUND_UNREPLICABLE} UINT; (*Interne Variable*)
		aInputArguments : {REDUND_UNREPLICABLE} ARRAY[0..MAX_INDEX_ARGUMENTS] OF UAMethodArgument; (*Interne Variable*)
		aOutputArguments : {REDUND_UNREPLICABLE} ARRAY[0..MAX_INDEX_ARGUMENTS] OF UAMethodArgument; (*Interne Variable*)
		eStep : {REDUND_UNREPLICABLE} DINT; (*Step-Nummer für die interne Schrittkette*)
		fbUA_MethodCall : {REDUND_UNREPLICABLE} UA_MethodCall; (*Interner FB*)
	END_VAR
END_FUNCTION_BLOCK

FUNCTION BrbUaRcGetSrvNamespace : UINT (*Gibt den Server-Namespace aufgrund des DatObj-NamespaceIndex zurück*) (*$GROUP=User,$CAT=User,$GROUPICON=User.png,$CATICON=User.png*)
	VAR_INPUT
		pRunClient : BrbUaRunClient_TYP; (*Zeiger auf die RunClient-Struktur*)
		nDatObjNamespaceIndex : UINT; (*0-basierter Index des Namespaces im Datenobjekt*)
		pServerNamespace : BrbUaRcNamespace_TYP; (*Zeiger auf die zu füllende Struktur*)
	END_VAR
END_FUNCTION

FUNCTION BrbUaRcGetNodeHandle : UINT (*Gibt einen ermittelten NodeHandle zurück*) (*$GROUP=User,$CAT=User,$GROUPICON=User.png,$CATICON=User.png*)
	VAR_INPUT
		pRunClient : BrbUaRunClient_TYP; (*Zeiger auf die RunClient-Struktur*)
		nNodeHandleIndex : UINT; (*0-basierter Index des NodeHandles*)
		pNodeHandle : BrbUaRcNodeHandle_TYP; (*Zeiger auf die zu füllende Struktur*)
	END_VAR
END_FUNCTION

FUNCTION BrbUaRcGetReadBlock : UINT (*Gibt einen ermittelten ReadBlock zurück*) (*$GROUP=User,$CAT=User,$GROUPICON=User.png,$CATICON=User.png*)
	VAR_INPUT
		pRunClient : BrbUaRunClient_TYP; (*Zeiger auf die RunClient-Struktur*)
		nReadBlockIndex : UINT; (*0-basierter Index des ReadBlocks*)
		pReadBlock : BrbUaRcReadBlock_TYP; (*Zeiger auf die zu füllende Struktur*)
		pReadBlockIntern : BrbUaRcReadBlockIntern_TYP; (*Zeiger auf die optional zu füllende, interne Struktur*)
	END_VAR
END_FUNCTION

FUNCTION BrbUaRcGetReadItem : UINT (*Gibt ein ermitteltes ReadItem zurück*) (*$GROUP=User,$CAT=User,$GROUPICON=User.png,$CATICON=User.png*)
	VAR_INPUT
		pRunClient : BrbUaRunClient_TYP; (*Zeiger auf die RunClient-Struktur*)
		nReadBlockIndex : UINT; (*0-basierter Index des ReadBlocks*)
		nReadItemIndex : UINT; (*0-basierter Index des ReadItems*)
		pReadItem : BrbUaRcReadItem_TYP; (*Zeiger auf die zu füllende Struktur*)
	END_VAR
END_FUNCTION

FUNCTION BrbUaRcGetWriteBlock : UINT (*Gibt einen ermittelten ReadBlock zurück*) (*$GROUP=User,$CAT=User,$GROUPICON=User.png,$CATICON=User.png*)
	VAR_INPUT
		pRunClient : BrbUaRunClient_TYP; (*Zeiger auf die RunClient-Struktur*)
		nWriteBlockIndex : UINT; (*0-basierter Index des WriteBlocks*)
		pWriteBlock : BrbUaRcWriteBlock_TYP; (*Zeiger auf die zu füllende Struktur*)
		pWriteBlockIntern : BrbUaRcWriteBlockIntern_TYP; (*Zeiger auf die optional zu füllende, interne Struktur*)
	END_VAR
END_FUNCTION

FUNCTION BrbUaRcGetWriteItem : UINT (*Gibt ein ermitteltes ReadItem zurück*) (*$GROUP=User,$CAT=User,$GROUPICON=User.png,$CATICON=User.png*)
	VAR_INPUT
		pRunClient : BrbUaRunClient_TYP; (*Zeiger auf die RunClient-Struktur*)
		nWriteBlockIndex : UINT; (*0-basierter Index des WriteBlocks*)
		nWriteItemIndex : UINT; (*0-basierter Index des WriteItems*)
		pWriteItem : BrbUaRcWriteItem_TYP; (*Zeiger auf die zu füllende Struktur*)
	END_VAR
END_FUNCTION

FUNCTION BrbUaRcGetMethod : UINT (*Gibt eine ermittelte Methode zuück*) (*$GROUP=User,$CAT=User,$GROUPICON=User.png,$CATICON=User.png*)
	VAR_INPUT
		pRunClient : BrbUaRunClient_TYP; (*Zeiger auf die RunClient-Struktur*)
		nMethodIndex : UINT; (*0-basierter Index der Method*)
		pMethod : BrbUaRcMethod_TYP; (*Zeiger auf die zu füllende Struktur*)
		pMethodIntern : BrbUaRcMethodIntern_TYP; (*Zeiger auf die optional zu füllende, interne Struktur*)
	END_VAR
END_FUNCTION

FUNCTION BrbUaRcGetArgument : UINT (*Gibt ein ermitteltes ReadItem zurück*) (*$GROUP=User,$CAT=User,$GROUPICON=User.png,$CATICON=User.png*)
	VAR_INPUT
		pRunClient : BrbUaRunClient_TYP; (*Zeiger auf die RunClient-Struktur*)
		nMethodIndex : UINT; (*0-basierter Index der Method*)
		bOutput : BOOL; (*0=Eingangs-Argument, 1=Ausgangs-Argument*)
		nArgumentIndex : UINT; (*0-basierter Index des Arguments*)
		pArgument : UAMethodArgument; (*Zeiger auf die zu füllende Struktur*)
	END_VAR
END_FUNCTION

FUNCTION BrbUaRcGetSubscription : UINT (*Gibt eine ermittelte Subscription zurück*) (*$GROUP=User,$CAT=User,$GROUPICON=User.png,$CATICON=User.png*)
	VAR_INPUT
		pRunClient : BrbUaRunClient_TYP; (*Zeiger auf die RunClient-Struktur*)
		nSubscriptionIndex : UINT; (*0-basierter Index der Subscription*)
		pSubscription : BrbUaRcSubscription_TYP; (*Zeiger auf die zu füllende Struktur*)
		pSubscriptionIntern : BrbUaRcSubscriptionIntern_TYP; (*Zeiger auf die optional zu füllende, interne Struktur*)
	END_VAR
END_FUNCTION

{REDUND_UNREPLICABLE} FUNCTION_BLOCK BrbUaRcSetSubscription (*Ändert die Parameter einer Subscription*) (*$GROUP=User,$CAT=User,$GROUPICON=User.png,$CATICON=User.png*)
	VAR_INPUT
		pRunClient : REFERENCE TO BrbUaRunClient_TYP; (*Zeiger auf die RunClient-Struktur*)
		nSubscriptionIndex : {REDUND_UNREPLICABLE} UINT; (*0-basierter Index der Subscription*)
		pSubscription : REFERENCE TO BrbUaRcSubscription_TYP; (*Zeiger auf die zu ändernden Werte*)
	END_VAR
	VAR_OUTPUT
		nStatus : {REDUND_UNREPLICABLE} DINT; (*Fub-Status*)
		bPublished : {REDUND_UNREPLICABLE} BOOL; (*Daten veröffentlicht seit dem letzten Aufruf*)
		nErrorId : {REDUND_UNREPLICABLE} DWORD; (*OpcUa-Fehler-Status*)
		sErrorId : {REDUND_UNREPLICABLE} STRING[80]; (*OpcUa-Fehler-Text*)
	END_VAR
	VAR
		eStep : {REDUND_UNREPLICABLE} DINT; (*Step-Nummer für die interne Schrittkette*)
		fbUA_SubscriptionOperate : {REDUND_UNREPLICABLE} UA_SubscriptionOperate; (*Interner FB*)
		tPublishingInterval : {REDUND_UNREPLICABLE} TIME; (*Interne Variable*)
	END_VAR
END_FUNCTION_BLOCK

FUNCTION BrbUaRcGetMonitoredItem : UINT (*Gibt ein ermitteltes MonitoredItem zurück*) (*$GROUP=User,$CAT=User,$GROUPICON=User.png,$CATICON=User.png*)
	VAR_INPUT
		pRunClient : BrbUaRunClient_TYP; (*Zeiger auf die RunClient-Struktur*)
		nSubscriptionIndex : UINT; (*0-basierter Index der Subscription*)
		nMonitoredItemIndex : UINT; (*0-basierter Index des MonitoredItems*)
		pMonitoredItem : BrbUaRcMonitoredItem_TYP; (*Zeiger auf die zu füllende Struktur*)
	END_VAR
END_FUNCTION

FUNCTION_BLOCK BrbUaRcSetMonitoredItem (*Ändert die Parameter eines MonitoredItems*) (*$GROUP=User,$CAT=User,$GROUPICON=User.png,$CATICON=User.png*)
	VAR_INPUT
		pRunClient : REFERENCE TO BrbUaRunClient_TYP; (*Zeiger auf die RunClient-Struktur*)
		nSubscriptionIndex : {REDUND_UNREPLICABLE} UINT; (*0-basierter Index der Subscription*)
		nMonitoredItemIndex : {REDUND_UNREPLICABLE} UINT; (*0-basierter Index des MonitoredItems*)
		pMonitoringSettings : REFERENCE TO UAMonitoringSettings; (*Zeiger auf die zu ändernden Werte*)
	END_VAR
	VAR_OUTPUT
		nStatus : {REDUND_UNREPLICABLE} DINT; (*Fub-Status*)
		bValueChanged : {REDUND_UNREPLICABLE} BOOL; (*Der Wert der überwachten Variable hat sich geändert*)
		dtTimestamp : {REDUND_UNREPLICABLE} DATE_AND_TIME; (*Zeitstempel der Änderung*)
		nErrorId : {REDUND_UNREPLICABLE} DWORD; (*OpcUa-Fehler-Status*)
		sErrorId : {REDUND_UNREPLICABLE} STRING[80]; (*OpcUa-Fehler-Text*)
	END_VAR
	VAR
		eStep : {REDUND_UNREPLICABLE} DINT; (*Step-Nummer für die interne Schrittkette*)
		fbUA_MonitoredItemOperate : {REDUND_UNREPLICABLE} UA_MonitoredItemOperate; (*Interner FB*)
		MonitoredItemIntern : BrbUaRcMonitoredItem_TYP; (*Interne Variable*)
	END_VAR
END_FUNCTION_BLOCK

FUNCTION BrbUaRcGetMiValueChanged : BOOL (*Gibt das ValueChanged-Flag eines MonitoredItems zurück und löscht es optional*) (*$GROUP=User,$CAT=User,$GROUPICON=User.png,$CATICON=User.png*)
	VAR_INPUT
		pRunClient : BrbUaRunClient_TYP; (*Zeiger auf die RunClient-Struktur*)
		nSubscriptionIndex : UINT; (*0-basierter Index der Subscription*)
		nMonitoredItemIndex : UINT; (*0-basierter Index des MonitoredItems*)
		bClear : BOOL; (*1=Flag löschen*)
	END_VAR
END_FUNCTION

FUNCTION BrbUaRcGetMiRemainingValueCount : UINT (*Gibt den RemainingValue-Zähler eines MonitoredItems zurück*) (*$GROUP=User,$CAT=User,$GROUPICON=User.png,$CATICON=User.png*)
	VAR_INPUT
		pRunClient : BrbUaRunClient_TYP; (*Zeiger auf die RunClient-Struktur*)
		nSubscriptionIndex : UINT; (*0-basierter Index der Subscription*)
		nMonitoredItemIndex : UINT; (*0-basierter Index des MonitoredItems*)
	END_VAR
END_FUNCTION

FUNCTION BrbUaRcGetEventItem : UINT (*Gibt ein ermitteltes EventItem zurück*) (*$GROUP=User,$CAT=User,$GROUPICON=User.png,$CATICON=User.png*)
	VAR_INPUT
		pRunClient : BrbUaRunClient_TYP; (*Zeiger auf die RunClient-Struktur*)
		nSubscriptionIndex : UINT; (*0-basierter Index der Subscription*)
		nEventItemIndex : UINT; (*0-basierter Index des EventItems*)
		pEventItem : BrbUaRcEventItem_TYP; (*Zeiger auf die zu füllende Struktur*)
		pEventItemIntern : BrbUaRcEventItemIntern_TYP; (*Zeiger auf die optional zu füllende, interne Struktur*)
	END_VAR
END_FUNCTION

FUNCTION BrbUaRcGetEventItemReceived : BOOL (*Gibt zurück, ob ein Event empfangen wurde*) (*$GROUP=User,$CAT=User,$GROUPICON=User.png,$CATICON=User.png*)
	VAR_INPUT
		pRunClient : BrbUaRunClient_TYP; (*Zeiger auf die RunClient-Struktur*)
		nSubscriptionIndex : UINT; (*0-basierter Index der Subscription*)
		nEventItemIndex : UINT; (*0-basierter Index des EventItems*)
	END_VAR
END_FUNCTION

FUNCTION BrbUaRcGetEventItemReceiveCount : UDINT (*Gibt zurück, wie oft ein Event empfangen wurde*) (*$GROUP=User,$CAT=User,$GROUPICON=User.png,$CATICON=User.png*)
	VAR_INPUT
		pRunClient : BrbUaRunClient_TYP; (*Zeiger auf die RunClient-Struktur*)
		nSubscriptionIndex : UINT; (*0-basierter Index der Subscription*)
		nEventItemIndex : UINT; (*0-basierter Index des EventItems*)
	END_VAR
END_FUNCTION

FUNCTION BrbUaRcGetEventField : UINT (*Gibt ein ermitteltes EventField zurück*) (*$GROUP=User,$CAT=User,$GROUPICON=User.png,$CATICON=User.png*)
	VAR_INPUT
		pRunClient : BrbUaRunClient_TYP; (*Zeiger auf die RunClient-Struktur*)
		nSubscriptionIndex : UINT; (*0-basierter Index der Subscription*)
		nEventItemIndex : UINT; (*0-basierter Index des EventItems*)
		nEventFieldIndex : UINT; (*0-basierter Index des EventFields*)
		pEventField : BrbUaRcEventField_TYP; (*Zeiger auf die zu füllende Struktur*)
	END_VAR
END_FUNCTION

FUNCTION BrbUaRcMonitor : UINT (*Zeigt die Inhalte des internen Speichers*) (*$GROUP=User,$CAT=User,$GROUPICON=User.png,$CATICON=User.png*)
	VAR_INPUT
		pRunClient : BrbUaRunClient_TYP; (*Zeiger auf die RunClient-Struktur*)
		pMonitor : BrbUaRcMonitor_TYP; (*Zeiger auf die Monitor-Struktur*)
	END_VAR
END_FUNCTION
(*Server - Methods*)

FUNCTION BrbUaSrvHandleMethod : DWORD (*Behandelt einen Methoden-Aufruf*) (*$GROUP=User,$CAT=User,$GROUPICON=User.png,$CATICON=User.png*)
	VAR_INPUT
		pMethod : BrbUaSrvMethod_TYP; (*Zeiger auf die Methode*)
	END_VAR
END_FUNCTION

FUNCTION BrbUaSrvGetMethodOperateText : DWORD (*Gibt den Text einer MethodOperateAction zurück*) (*$GROUP=User,$CAT=User,$GROUPICON=User.png,$CATICON=User.png*)
	VAR_INPUT
		eAction : UaMethodOperateAction; (*Angabe der Aktion*)
		pActionText : STRING[0]; (*Zeiger auf den String*)
		nActionTextSize : UDINT; (*Größe des Strings*)
	END_VAR
END_FUNCTION
(*Server - RunServer*)

{REDUND_UNREPLICABLE} FUNCTION_BLOCK BrbUaRunServerInit (*Initialisiert eine Server-Instanz*) (*$GROUP=User,$CAT=User,$GROUPICON=User.png,$CATICON=User.png*)
	VAR_INPUT
		pRunServer : REFERENCE TO BrbUaRunServer_TYP; (*Zeiger auf die RunServer-Struktur*)
	END_VAR
	VAR_OUTPUT
		nStatus : {REDUND_UNREPLICABLE} UINT; (*Fub-Status*)
	END_VAR
	VAR
		eStep : {REDUND_UNREPLICABLE} DINT; (*Step-Nummer für die interne Schrittkette*)
		fbDatObjInfo : {REDUND_UNREPLICABLE} DatObjInfo; (*Interner FB*)
		fbDatObjRead : {REDUND_UNREPLICABLE} DatObjRead; (*Interner FB*)
		nAllocStatus : {REDUND_UNREPLICABLE} UINT; (*Interne Variable*)
		nNamespaceIndex : {REDUND_UNREPLICABLE} DINT; (*Interne Variable*)
		nEventIndex : {REDUND_UNREPLICABLE} DINT; (*Interne Variable*)
		nEventFieldIndex : {REDUND_UNREPLICABLE} DINT; (*Interne Variable*)
		nLoopIndex : {REDUND_UNREPLICABLE} UINT; (*Interne Variable*)
		sLine : {REDUND_UNREPLICABLE} STRING[1024]; (*Interne Variable*)
		nLineLen : {REDUND_UNREPLICABLE} UDINT; (*Interne Variable*)
		sValue : {REDUND_UNREPLICABLE} STRING[1024]; (*Interne Variable*)
		nValue : {REDUND_UNREPLICABLE} DINT; (*Interne Variable*)
		rValue : {REDUND_UNREPLICABLE} REAL; (*Interne Variable*)
		sVarName : {REDUND_UNREPLICABLE} STRING[nBRBUA_VARNAME_TEXT_CHAR_MAX]; (*Interne Variable*)
	END_VAR
END_FUNCTION_BLOCK

{REDUND_UNREPLICABLE} FUNCTION_BLOCK BrbUaRunServerCyclic (*Behandelt eine Server-Instanz*) (*$GROUP=User,$CAT=User,$GROUPICON=User.png,$CATICON=User.png*)
	VAR_INPUT
		pRunServer : REFERENCE TO BrbUaRunServer_TYP; (*Zeiger auf die RunServer-Struktur*)
	END_VAR
	VAR_OUTPUT
		nStatus : {REDUND_UNREPLICABLE} UINT; (*Fub-Status*)
	END_VAR
	VAR
		eStep : {REDUND_UNREPLICABLE} DINT; (*Step-Nummer für die interne Schrittkette*)
		fbUaSrv_GetNamespaceIndex : {REDUND_UNREPLICABLE} UaSrv_GetNamespaceIndex; (*Interner FB*)
		nNamespaceIndex : {REDUND_UNREPLICABLE} DINT; (*Interne Variable*)
		nLoopIndex : {REDUND_UNREPLICABLE} UINT; (*Interne Variable*)
		nEventIndex : {REDUND_UNREPLICABLE} DINT; (*Interne Variable*)
		nEventFieldIndex : {REDUND_UNREPLICABLE} DINT; (*Interne Variable*)
	END_VAR
END_FUNCTION_BLOCK

{REDUND_UNREPLICABLE} FUNCTION_BLOCK BrbUaRunServerExit (*Exilisiert eine Server-Instanz*) (*$GROUP=User,$CAT=User,$GROUPICON=User.png,$CATICON=User.png*)
	VAR_INPUT
		pRunServer : REFERENCE TO BrbUaRunServer_TYP; (*Zeiger auf die RunServer-Struktur*)
	END_VAR
	VAR_OUTPUT
		nStatus : {REDUND_UNREPLICABLE} UINT; (*Fub-Status*)
	END_VAR
	VAR
		eStep : {REDUND_UNREPLICABLE} DINT; (*Step-Nummer für die interne Schrittkette*)
		nEventIndex : {REDUND_UNREPLICABLE} DINT; (*Interne Variable*)
		nFreeStatus : {REDUND_UNREPLICABLE} UINT; (*Interne Variable*)
	END_VAR
END_FUNCTION_BLOCK

FUNCTION_BLOCK BrbUaRsFireEvent (*Liest eine ReadBlock vom Server*) (*$GROUP=User,$CAT=User,$GROUPICON=User.png,$CATICON=User.png*)
	VAR_INPUT
		pRunServer : REFERENCE TO BrbUaRunServer_TYP; (*Zeiger auf die RunServer-Struktur*)
		nEventIndex : {REDUND_UNREPLICABLE} UINT; (*0-basierter Index des Events*)
	END_VAR
	VAR_OUTPUT
		bInit : {REDUND_UNREPLICABLE} BOOL; (*Vor dem Fire für einen Zyklus auf 1*)
		nStatus : {REDUND_UNREPLICABLE} UINT; (*Fub-Status*)
		nErrorId : {REDUND_UNREPLICABLE} DWORD; (*OpcUa-Fehler-Status*)
		sErrorId : {REDUND_UNREPLICABLE} STRING[nBRBUA_STATUS_TEXT_CHAR_MAX]; (*OpcUa-Fehler-Text*)
		nFireCount : UDINT; (*Anzahl der gefeuerten Events*)
	END_VAR
	VAR
		eStep : {REDUND_UNREPLICABLE} DINT; (*Step-Nummer für die interne Schrittkette*)
		fbUaSrv_FireEvent : {REDUND_UNREPLICABLE} UaSrv_FireEvent; (*Interner FB*)
	END_VAR
END_FUNCTION_BLOCK

FUNCTION BrbUaRsGetNamespace : UINT (*Gibt den Server-Namespace aufgrund des DataObjekt-NamespaceIndex zurück*) (*$GROUP=User,$CAT=User,$GROUPICON=User.png,$CATICON=User.png*)
	VAR_INPUT
		pRunServer : BrbUaRunServer_TYP; (*Zeiger auf die RunClient-Struktur*)
		nDatObjNamespaceIndex : UINT; (*0-basierter Index des Namespaces im Datenobjekt*)
		pServerNamespace : BrbUaRsNamespace_TYP; (*Zeiger auf die zu füllende Struktur*)
	END_VAR
END_FUNCTION

FUNCTION BrbUaRsGetEvent : UINT (*Gibt ein ermitteltes Event zurück*) (*$GROUP=User,$CAT=User,$GROUPICON=User.png,$CATICON=User.png*)
	VAR_INPUT
		pRunServer : BrbUaRunServer_TYP; (*Zeiger auf die RunClient-Struktur*)
		nEventIndex : UINT; (*0-basierter Index des Events*)
		pEvent : BrbUaRsEvent_TYP; (*Zeiger auf die zu füllende Struktur*)
		pEventIntern : BrbUaRsEventIntern_TYP; (*Zeiger auf die optional zu füllende, interne Struktur*)
	END_VAR
END_FUNCTION

FUNCTION BrbUaRsGetEventField : UINT (*Gibt ein ermitteltes Field zurück*) (*$GROUP=User,$CAT=User,$GROUPICON=User.png,$CATICON=User.png*)
	VAR_INPUT
		pRunServer : BrbUaRunServer_TYP; (*Zeiger auf die RunClient-Struktur*)
		nEventIndex : UINT; (*0-basierter Index des Events*)
		nEventFieldIndex : UINT; (*0-basierter Index des Fields*)
		pEventField : UaSrv_FireEventFieldType; (*Zeiger auf die zu füllende Struktur*)
	END_VAR
END_FUNCTION

FUNCTION BrbUaRsMonitor : UINT (*Zeigt die Inhalte des internen Speichers*) (*$GROUP=User,$CAT=User,$GROUPICON=User.png,$CATICON=User.png*)
	VAR_INPUT
		pRunServer : BrbUaRunServer_TYP; (*Zeiger auf die RunServer-Struktur*)
		pMonitor : BrbUaRsMonitor_TYP; (*Zeiger auf die Monitor-Struktur*)
	END_VAR
END_FUNCTION
```
